LIN {X 0,Y 532.498,Z 413.718,A -85,B 0,C 180,E1 -4445.914,E2 -4445.914} C_VEL
LIN {X 0,Y 531.12,Z 406.108,A -85,B 0,C 180,E1 -4447.734,E2 -4447.734} C_VEL
LIN {X 0,Y 530.969,Z 405.349,A -85,B 0,C 180,E1 -4447.987,E2 -4447.987} C_VEL
LIN {X 0,Y 531.028,Z 405.342,A -85,B 0,C 180,E1 -4450.429,E2 -4450.429} C_VEL
LIN {X 0,Y 530.956,Z 405.351,A -85,B 0,C 180,E1 -4453.495,E2 -4453.495} C_VEL
LIN {X 0,Y 530.968,Z 405.348,A -85,B 0,C 180,E1 -4456.506,E2 -4456.506} C_VEL
LIN {X 0,Y 530.991,Z 405.345,A -85,B 0,C 180,E1 -4458.976,E2 -4458.976} C_VEL
LIN {X 0,Y 530.962,Z 405.348,A -85,B 0,C 180,E1 -4461.53,E2 -4461.53} C_VEL
LIN {X 0,Y 530.978,Z 405.348,A -85,B 0,C 180,E1 -4464.382,E2 -4464.382} C_VEL
LIN {X 0,Y 530.968,Z 405.345,A -85,B 0,C 180,E1 -4467.133,E2 -4467.133} C_VEL
LIN {X 0,Y 530.971,Z 405.348,A -85,B 0,C 180,E1 -4469.803,E2 -4469.803} C_VEL
LIN {X 0,Y 531.02,Z 405.341,A -85,B 0,C 180,E1 -4472.466,E2 -4472.466} C_VEL
LIN {X 0,Y 531.011,Z 405.342,A -85,B 0,C 180,E1 -4474.943,E2 -4474.943} C_VEL
LIN {X 0,Y 530.974,Z 405.347,A -85,B 0,C 180,E1 -4478.247,E2 -4478.247} C_VEL
LIN {X 0,Y 530.998,Z 405.345,A -85,B 0,C 180,E1 -4480.677,E2 -4480.677} C_VEL
LIN {X 0,Y 530.989,Z 405.344,A -85,B 0,C 180,E1 -4483.071,E2 -4483.071} C_VEL
LIN {X 0,Y 531.022,Z 405.34,A -85,B 0,C 180,E1 -4485.436,E2 -4485.436} C_VEL
LIN {X 0,Y 531.051,Z 405.337,A -85,B 0,C 180,E1 -4488.55,E2 -4488.55} C_VEL
LIN {X 0,Y 531.04,Z 405.34,A -85,B 0,C 180,E1 -4491.629,E2 -4491.629} C_VEL
LIN {X 0,Y 531.125,Z 405.329,A -85,B 0,C 180,E1 -4494.685,E2 -4494.685} C_VEL
LIN {X 0,Y 531.145,Z 405.325,A -85,B 0,C 180,E1 -4497.725,E2 -4497.725} C_VEL
LIN {X 0,Y 531.157,Z 405.323,A -85,B 0,C 180,E1 -4500.758,E2 -4500.758} C_VEL
LIN {X 0,Y 531.107,Z 405.328,A -85,B 0,C 180,E1 -4503.034,E2 -4503.034} C_VEL
LIN {X 0,Y 531.085,Z 405.333,A -85,B 0,C 180,E1 -4506.077,E2 -4506.077} C_VEL
LIN {X 0,Y 531.035,Z 405.339,A -85,B 0,C 180,E1 -4509.138,E2 -4509.138} C_VEL
LIN {X 0,Y 531.044,Z 405.339,A -85,B 0,C 180,E1 -4512.225,E2 -4512.225} C_VEL
LIN {X 0,Y 530.998,Z 405.344,A -85,B 0,C 180,E1 -4515.35,E2 -4515.35} C_VEL
LIN {X 0,Y 530.993,Z 405.345,A -85,B 0,C 180,E1 -4518.521,E2 -4518.521} C_VEL
LIN {X 0,Y 531.005,Z 405.343,A -85,B 0,C 180,E1 -4520.938,E2 -4520.938} C_VEL
LIN {X 0,Y 530.983,Z 405.346,A -85,B 0,C 180,E1 -4524.225,E2 -4524.225} C_VEL
LIN {X 0,Y 531.007,Z 405.341,A -85,B 0,C 180,E1 -4526.744,E2 -4526.744} C_VEL
LIN {X 0,Y 530.984,Z 405.345,A -85,B 0,C 180,E1 -4529.323,E2 -4529.323} C_VEL
LIN {X 0,Y 530.973,Z 405.347,A -85,B 0,C 180,E1 -4532.101,E2 -4532.101} C_VEL
LIN {X 0,Y 530.988,Z 405.345,A -85,B 0,C 180,E1 -4534.854,E2 -4534.854} C_VEL
LIN {X 0,Y 530.97,Z 405.347,A -85,B 0,C 180,E1 -4537.508,E2 -4537.508} C_VEL
LIN {X 0,Y 530.984,Z 405.345,A -85,B 0,C 180,E1 -4540.433,E2 -4540.433} C_VEL
LIN {X 0,Y 530.97,Z 405.348,A -85,B 0,C 180,E1 -4543.495,E2 -4543.495} C_VEL
LIN {X 0,Y 530.967,Z 405.348,A -85,B 0,C 180,E1 -4543.57,E2 -4543.57} C_VEL
LIN {X 0,Y 530.294,Z 405.432,A -85,B 0,C 180,E1 -4544.203,E2 -4544.203} C_VEL
LIN {X 0,Y 527.447,Z 405.786,A -85,B 0,C 180,E1 -4545.232,E2 -4545.232} C_VEL
LIN {X 0,Y 525.044,Z 406.087,A -85,B 0,C 180,E1 -4546.061,E2 -4546.061} C_VEL
LIN {X 0,Y 524.011,Z 406.214,A -85,B 0,C 180,E1 -4546.7,E2 -4546.7} C_VEL
LIN {X 0,Y 523.926,Z 406.224,A -85,B 0,C 180,E1 -4546.917,E2 -4546.917} C_VEL
LIN {X 0,Y 523.951,Z 406.223,A -85,B 0,C 180,E1 -4549.921,E2 -4549.921} C_VEL
LIN {X 0,Y 523.914,Z 406.224,A -85,B 0,C 180,E1 -4552.868,E2 -4552.868} C_VEL
LIN {X 0,Y 523.947,Z 406.223,A -85,B 0,C 180,E1 -4555.711,E2 -4555.711} C_VEL
LIN {X 0,Y 523.938,Z 406.224,A -85,B 0,C 180,E1 -4558.457,E2 -4558.457} C_VEL
LIN {X 0,Y 523.948,Z 406.222,A -85,B 0,C 180,E1 -4561.126,E2 -4561.126} C_VEL
LIN {X 0,Y 523.988,Z 406.218,A -85,B 0,C 180,E1 -4563.981,E2 -4563.981} C_VEL
LIN {X 0,Y 523.931,Z 406.224,A -85,B 0,C 180,E1 -4566.271,E2 -4566.271} C_VEL
LIN {X 0,Y 523.951,Z 406.221,A -85,B 0,C 180,E1 -4568.767,E2 -4568.767} C_VEL
LIN {X 0,Y 523.958,Z 406.22,A -85,B 0,C 180,E1 -4571.221,E2 -4571.221} C_VEL
LIN {X 0,Y 523.94,Z 406.223,A -85,B 0,C 180,E1 -4573.639,E2 -4573.639} C_VEL
LIN {X 0,Y 523.944,Z 406.224,A -85,B 0,C 180,E1 -4576.028,E2 -4576.028} C_VEL
LIN {X 0,Y 524.018,Z 406.214,A -85,B 0,C 180,E1 -4578.394,E2 -4578.394} C_VEL
LIN {X 0,Y 523.991,Z 406.288,A -85,B 0,C 180,E1 -4580.105,E2 -4580.105} C_VEL
LIN {X 0,Y 525.17,Z 411.277,A -85,B 0,C 180,E1 -4580.37,E2 -4580.37} C_VEL
LIN {X 0,Y 524.954,Z 423.401,A -85,B 0,C 180,E1 -4581.047,E2 -4581.047} C_VEL
LIN {X 0,Y 524.619,Z 435.388,A -85,B 0,C 180,E1 -4581.914,E2 -4581.914} C_VEL
LIN {X 0,Y 524.34,Z 445.661,A -85,B 0,C 180,E1 -4582.859,E2 -4582.859} C_VEL
LIN {X 0,Y 524.058,Z 454.306,A -85,B 0,C 180,E1 -4583.841,E2 -4583.841} C_VEL
LIN {X 0,Y 523.918,Z 461.363,A -85,B 0,C 180,E1 -4584.805,E2 -4584.805} C_VEL
LIN {X 0,Y 523.73,Z 468.234,A -85,B 0,C 180,E1 -4585.96,E2 -4585.96} C_VEL
LIN {X 0,Y 523.563,Z 474.542,A -85,B 0,C 180,E1 -4587.307,E2 -4587.307} C_VEL
LIN {X 0,Y 523.457,Z 479.837,A -85,B 0,C 180,E1 -4588.846,E2 -4588.846} C_VEL
LIN {X 0,Y 523.3,Z 482.596,A -85,B 0,C 180,E1 -4590,E2 -4590} C_VEL
LIN {X 0,Y 523.287,Z 483.993,A -85,B 0,C 180,E1 -4590.77,E2 -4590.77} C_VEL
LIN {X 0,Y 523.345,Z 485.482,A -85,B 0,C 180,E1 -4592.309,E2 -4592.309} C_VEL
LIN {X 0,Y 523.39,Z 485.664,A -85,B 0,C 180,E1 -4593.079,E2 -4593.079} C_VEL
LIN {X 0,Y 523.432,Z 485.43,A -85,B 0,C 180,E1 -4593.85,E2 -4593.85} C_VEL
LIN {X 0,Y 523.387,Z 483.874,A -85,B 0,C 180,E1 -4595.394,E2 -4595.394} C_VEL
LIN {X 0,Y 523.454,Z 480.665,A -85,B 0,C 180,E1 -4596.941,E2 -4596.941} C_VEL
LIN {X 0,Y 523.508,Z 477.124,A -85,B 0,C 180,E1 -4598.104,E2 -4598.104} C_VEL
LIN {X 0,Y 523.584,Z 472.411,A -85,B 0,C 180,E1 -4599.269,E2 -4599.269} C_VEL
LIN {X 0,Y 523.77,Z 466.518,A -85,B 0,C 180,E1 -4600.437,E2 -4600.437} C_VEL
LIN {X 0,Y 523.901,Z 459.174,A -85,B 0,C 180,E1 -4601.609,E2 -4601.609} C_VEL
LIN {X 0,Y 524.181,Z 449.879,A -85,B 0,C 180,E1 -4602.781,E2 -4602.781} C_VEL
LIN {X 0,Y 524.418,Z 440.224,A -85,B 0,C 180,E1 -4603.762,E2 -4603.762} C_VEL
LIN {X 0,Y 524.739,Z 430.634,A -85,B 0,C 180,E1 -4604.544,E2 -4604.544} C_VEL
LIN {X 0,Y 525.04,Z 420.234,A -85,B 0,C 180,E1 -4605.236,E2 -4605.236} C_VEL
LIN {X 0,Y 525.018,Z 410.197,A -85,B 0,C 180,E1 -4605.778,E2 -4605.778} C_VEL
LIN {X 0,Y 523.966,Z 406.223,A -85,B 0,C 180,E1 -4606.01,E2 -4606.01} C_VEL
LIN {X 0,Y 523.953,Z 406.22,A -85,B 0,C 180,E1 -4608.779,E2 -4608.779} C_VEL
LIN {X 0,Y 523.951,Z 406.215,A -85,B 0,C 180,E1 -4611.233,E2 -4611.233} C_VEL
LIN {X 0,Y 523.931,Z 406.222,A -85,B 0,C 180,E1 -4614.572,E2 -4614.572} C_VEL
LIN {X 0,Y 523.952,Z 406.214,A -85,B 0,C 180,E1 -4617.133,E2 -4617.133} C_VEL
LIN {X 0,Y 523.948,Z 406.217,A -85,B 0,C 180,E1 -4619.756,E2 -4619.756} C_VEL
LIN {X 0,Y 523.938,Z 406.221,A -85,B 0,C 180,E1 -4622.45,E2 -4622.45} C_VEL
LIN {X 0,Y 523.938,Z 406.216,A -85,B 0,C 180,E1 -4625.226,E2 -4625.226} C_VEL
LIN {X 0,Y 523.921,Z 406.226,A -85,B 0,C 180,E1 -4628.102,E2 -4628.102} C_VEL
LIN {X 0,Y 523.944,Z 406.215,A -85,B 0,C 180,E1 -4631.092,E2 -4631.092} C_VEL
LIN {X 0,Y 523.942,Z 406.222,A -85,B 0,C 180,E1 -4634.228,E2 -4634.228} C_VEL
LIN {X 0,Y 523.926,Z 406.217,A -85,B 0,C 180,E1 -4636.833,E2 -4636.833} C_VEL
LIN {X 0,Y 523.947,Z 406.215,A -85,B 0,C 180,E1 -4638.908,E2 -4638.908} C_VEL
LIN {X 0,Y 523.92,Z 406.226,A -85,B 0,C 180,E1 -4641.898,E2 -4641.898} C_VEL
LIN {X 0,Y 523.929,Z 406.217,A -85,B 0,C 180,E1 -4644.911,E2 -4644.911} C_VEL
LIN {X 0,Y 523.94,Z 406.221,A -85,B 0,C 180,E1 -4647.68,E2 -4647.68} C_VEL
LIN {X 0,Y 523.959,Z 406.213,A -85,B 0,C 180,E1 -4650.676,E2 -4650.676} C_VEL
LIN {X 0,Y 523.978,Z 406.218,A -85,B 0,C 180,E1 -4653.728,E2 -4653.728} C_VEL
LIN {X 0,Y 523.917,Z 406.221,A -85,B 0,C 180,E1 -4656.27,E2 -4656.27} C_VEL
LIN {X 0,Y 523.95,Z 406.214,A -85,B 0,C 180,E1 -4658.767,E2 -4658.767} C_VEL
LIN {X 0,Y 523.953,Z 406.216,A -85,B 0,C 180,E1 -4661.221,E2 -4661.221} C_VEL
LIN {X 0,Y 523.934,Z 406.224,A -85,B 0,C 180,E1 -4663.639,E2 -4663.639} C_VEL
LIN {X 0,Y 523.944,Z 406.221,A -85,B 0,C 180,E1 -4666.028,E2 -4666.028} C_VEL
LIN {X 0,Y 524.031,Z 406.283,A -85,B 0,C 180,E1 -4668.148,E2 -4668.148} C_VEL
LIN {X 0,Y 525.077,Z 411.361,A -85,B 0,C 180,E1 -4668.418,E2 -4668.418} C_VEL
LIN {X 0,Y 524.956,Z 421.94,A -85,B 0,C 180,E1 -4669.002,E2 -4669.002} C_VEL
LIN {X 0,Y 524.603,Z 433.114,A -85,B 0,C 180,E1 -4669.775,E2 -4669.775} C_VEL
LIN {X 0,Y 524.321,Z 444.072,A -85,B 0,C 180,E1 -4670.744,E2 -4670.744} C_VEL
LIN {X 0,Y 524.042,Z 452.907,A -85,B 0,C 180,E1 -4671.711,E2 -4671.711} C_VEL
LIN {X 0,Y 523.887,Z 460.199,A -85,B 0,C 180,E1 -4672.678,E2 -4672.678} C_VEL
LIN {X 0,Y 523.758,Z 467.369,A -85,B 0,C 180,E1 -4673.837,E2 -4673.837} C_VEL
LIN {X 0,Y 523.529,Z 473.11,A -85,B 0,C 180,E1 -4674.994,E2 -4674.994} C_VEL
LIN {X 0,Y 523.508,Z 477.591,A -85,B 0,C 180,E1 -4676.151,E2 -4676.151} C_VEL
LIN {X 0,Y 523.467,Z 479.958,A -85,B 0,C 180,E1 -4676.921,E2 -4676.921} C_VEL
LIN {X 0,Y 523.309,Z 483.443,A -85,B 0,C 180,E1 -4678.461,E2 -4678.461} C_VEL
LIN {X 0,Y 523.283,Z 484.58,A -85,B 0,C 180,E1 -4679.23,E2 -4679.23} C_VEL
LIN {X 0,Y 523.278,Z 485.616,A -85,B 0,C 180,E1 -4680.769,E2 -4680.769} C_VEL
LIN {X 0,Y 523.295,Z 485.594,A -85,B 0,C 180,E1 -4681.539,E2 -4681.539} C_VEL
LIN {X 0,Y 523.395,Z 484.295,A -85,B 0,C 180,E1 -4683.079,E2 -4683.079} C_VEL
LIN {X 0,Y 523.441,Z 483.112,A -85,B 0,C 180,E1 -4683.849,E2 -4683.849} C_VEL
LIN {X 0,Y 523.41,Z 480.522,A -85,B 0,C 180,E1 -4685.007,E2 -4685.007} C_VEL
LIN {X 0,Y 523.523,Z 476.921,A -85,B 0,C 180,E1 -4686.165,E2 -4686.165} C_VEL
LIN {X 0,Y 523.596,Z 472.211,A -85,B 0,C 180,E1 -4687.326,E2 -4687.326} C_VEL
LIN {X 0,Y 523.761,Z 466.229,A -85,B 0,C 180,E1 -4688.488,E2 -4688.488} C_VEL
LIN {X 0,Y 523.913,Z 460.139,A -85,B 0,C 180,E1 -4689.458,E2 -4689.458} C_VEL
LIN {X 0,Y 524.125,Z 452.795,A -85,B 0,C 180,E1 -4690.429,E2 -4690.429} C_VEL
LIN {X 0,Y 524.38,Z 443.885,A -85,B 0,C 180,E1 -4691.402,E2 -4691.402} C_VEL
LIN {X 0,Y 524.656,Z 432.719,A -85,B 0,C 180,E1 -4692.376,E2 -4692.376} C_VEL
LIN {X 0,Y 524.959,Z 421.283,A -85,B 0,C 180,E1 -4693.155,E2 -4693.155} C_VEL
LIN {X 0,Y 524.995,Z 410.363,A -85,B 0,C 180,E1 -4693.746,E2 -4693.746} C_VEL
LIN {X 0,Y 524.004,Z 406.214,A -85,B 0,C 180,E1 -4693.97,E2 -4693.97} C_VEL
LIN {X 0,Y 523.962,Z 406.221,A -85,B 0,C 180,E1 -4697.163,E2 -4697.163} C_VEL
LIN {X 0,Y 523.977,Z 406.221,A -85,B 0,C 180,E1 -4700.41,E2 -4700.41} C_VEL
LIN {X 0,Y 523.915,Z 406.228,A -85,B 0,C 180,E1 -4702.893,E2 -4702.893} C_VEL
LIN {X 0,Y 523.989,Z 406.217,A -85,B 0,C 180,E1 -4706.02,E2 -4706.02} C_VEL
LIN {X 0,Y 523.944,Z 406.222,A -85,B 0,C 180,E1 -4708.874,E2 -4708.874} C_VEL
LIN {X 0,Y 523.925,Z 406.225,A -85,B 0,C 180,E1 -4711.544,E2 -4711.544} C_VEL
LIN {X 0,Y 523.937,Z 406.224,A -85,B 0,C 180,E1 -4714.29,E2 -4714.29} C_VEL
LIN {X 0,Y 523.91,Z 406.226,A -85,B 0,C 180,E1 -4717.132,E2 -4717.132} C_VEL
LIN {X 0,Y 523.941,Z 406.222,A -85,B 0,C 180,E1 -4720.13,E2 -4720.13} C_VEL
LIN {X 0,Y 523.928,Z 406.223,A -85,B 0,C 180,E1 -4723.166,E2 -4723.166} C_VEL
LIN {X 0,Y 523.939,Z 406.22,A -85,B 0,C 180,E1 -4725.772,E2 -4725.772} C_VEL
LIN {X 0,Y 523.945,Z 406.222,A -85,B 0,C 180,E1 -4728.908,E2 -4728.908} C_VEL
LIN {X 0,Y 523.983,Z 406.405,A -85,B 0,C 180,E1 -4731.781,E2 -4731.781} C_VEL
LIN {X 0,Y 525.435,Z 413.966,A -85,B 0,C 180,E1 -4733.678,E2 -4733.678} C_VEL
LIN {X 0,Y 525.524,Z 419.21,A -85,B 0,C 180,E1 -4734.896,E2 -4734.896} C_VEL
LIN {X 0,Y 525.11,Z 433.663,A -85,B 0,C 180,E1 -4738.085,E2 -4738.085} C_VEL
LIN {X 0,Y 524.935,Z 446.556,A -85,B 0,C 180,E1 -4740.832,E2 -4740.832} C_VEL
LIN {X 0,Y 524.742,Z 461.045,A -85,B 0,C 180,E1 -4743.812,E2 -4743.812} C_VEL
LIN {X 0,Y 524.523,Z 476.503,A -85,B 0,C 180,E1 -4746.926,E2 -4746.926} C_VEL
LIN {X 0,Y 524.282,Z 490.939,A -85,B 0,C 180,E1 -4749.777,E2 -4749.777} C_VEL
LIN {X 0,Y 524.177,Z 504.983,A -85,B 0,C 180,E1 -4752.504,E2 -4752.504} C_VEL
LIN {X 0,Y 523.941,Z 522.326,A -85,B 0,C 180,E1 -4755.83,E2 -4755.83} C_VEL
LIN {X 0,Y 523.852,Z 524.508,A -85,B 0,C 180,E1 -4756.248,E2 -4756.248} C_VEL
LIN {X 0,Y 525.46,Z 535.938,A -85,B 0,C 180,E1 -4756.513,E2 -4756.513} C_VEL
LIN {X 0,Y 525.206,Z 548.7,A -85,B 0,C 180,E1 -4756.9,E2 -4756.9} C_VEL
LIN {X 0,Y 524.979,Z 561.165,A -85,B 0,C 180,E1 -4757.435,E2 -4757.435} C_VEL
LIN {X 0,Y 524.711,Z 573.14,A -85,B 0,C 180,E1 -4758.113,E2 -4758.113} C_VEL
LIN {X 0,Y 524.458,Z 583.898,A -85,B 0,C 180,E1 -4758.893,E2 -4758.893} C_VEL
LIN {X 0,Y 524.169,Z 593.595,A -85,B 0,C 180,E1 -4759.767,E2 -4759.767} C_VEL
LIN {X 0,Y 523.93,Z 602.411,A -85,B 0,C 180,E1 -4760.737,E2 -4760.737} C_VEL
LIN {X 0,Y 523.724,Z 611.003,A -85,B 0,C 180,E1 -4761.9,E2 -4761.9} C_VEL
LIN {X 0,Y 523.575,Z 617.867,A -85,B 0,C 180,E1 -4763.061,E2 -4763.061} C_VEL
LIN {X 0,Y 523.544,Z 623.365,A -85,B 0,C 180,E1 -4764.222,E2 -4764.222} C_VEL
LIN {X 0,Y 523.361,Z 627.676,A -85,B 0,C 180,E1 -4765.378,E2 -4765.378} C_VEL
LIN {X 0,Y 523.443,Z 629.957,A -85,B 0,C 180,E1 -4766.151,E2 -4766.151} C_VEL
LIN {X 0,Y 523.367,Z 631.806,A -85,B 0,C 180,E1 -4766.921,E2 -4766.921} C_VEL
LIN {X 0,Y 523.334,Z 633.193,A -85,B 0,C 180,E1 -4767.691,E2 -4767.691} C_VEL
LIN {X 0,Y 523.25,Z 634.785,A -85,B 0,C 180,E1 -4769.23,E2 -4769.23} C_VEL
LIN {X 0,Y 523.246,Z 635,A -85,B 0,C 180,E1 -4770,E2 -4770} C_VEL
LIN {X 0,Y 523.274,Z 634.184,A -85,B 0,C 180,E1 -4771.539,E2 -4771.539} C_VEL
LIN {X 0,Y 523.334,Z 633.196,A -85,B 0,C 180,E1 -4772.309,E2 -4772.309} C_VEL
LIN {X 0,Y 523.367,Z 631.81,A -85,B 0,C 180,E1 -4773.079,E2 -4773.079} C_VEL
LIN {X 0,Y 523.441,Z 628.896,A -85,B 0,C 180,E1 -4774.235,E2 -4774.235} C_VEL
LIN {X 0,Y 523.464,Z 624.948,A -85,B 0,C 180,E1 -4775.393,E2 -4775.393} C_VEL
LIN {X 0,Y 523.523,Z 619.727,A -85,B 0,C 180,E1 -4776.581,E2 -4776.581} C_VEL
LIN {X 0,Y 523.665,Z 613.467,A -85,B 0,C 180,E1 -4777.713,E2 -4777.713} C_VEL
LIN {X 0,Y 523.857,Z 605.478,A -85,B 0,C 180,E1 -4778.875,E2 -4778.875} C_VEL
LIN {X 0,Y 524.085,Z 597.334,A -85,B 0,C 180,E1 -4779.845,E2 -4779.845} C_VEL
LIN {X 0,Y 524.36,Z 587.395,A -85,B 0,C 180,E1 -4780.815,E2 -4780.815} C_VEL
LIN {X 0,Y 524.647,Z 577.521,A -85,B 0,C 180,E1 -4781.592,E2 -4781.592} C_VEL
LIN {X 0,Y 524.881,Z 566.042,A -85,B 0,C 180,E1 -4782.308,E2 -4782.308} C_VEL
LIN {X 0,Y 525.095,Z 553.693,A -85,B 0,C 180,E1 -4782.906,E2 -4782.906} C_VEL
LIN {X 0,Y 525.356,Z 540.547,A -85,B 0,C 180,E1 -4783.367,E2 -4783.367} C_VEL
LIN {X 0,Y 525.221,Z 533.738,A -85,B 0,C 180,E1 -4783.542,E2 -4783.542} C_VEL
LIN {X 0,Y 523.852,Z 524.533,A -85,B 0,C 180,E1 -4783.752,E2 -4783.752} C_VEL
LIN {X 0,Y 524.05,Z 509.933,A -85,B 0,C 180,E1 -4786.558,E2 -4786.558} C_VEL
LIN {X 0,Y 524.265,Z 495.307,A -85,B 0,C 180,E1 -4789.377,E2 -4789.377} C_VEL
LIN {X 0,Y 524.466,Z 481.727,A -85,B 0,C 180,E1 -4792.037,E2 -4792.037} C_VEL
LIN {X 0,Y 524.666,Z 466.125,A -85,B 0,C 180,E1 -4795.169,E2 -4795.169} C_VEL
LIN {X 0,Y 524.892,Z 451.487,A -85,B 0,C 180,E1 -4798.163,E2 -4798.163} C_VEL
LIN {X 0,Y 525.061,Z 437.633,A -85,B 0,C 180,E1 -4801.058,E2 -4801.058} C_VEL
LIN {X 0,Y 525.301,Z 424.197,A -85,B 0,C 180,E1 -4803.953,E2 -4803.953} C_VEL
LIN {X 0,Y 525.529,Z 414.817,A -85,B 0,C 180,E1 -4806.045,E2 -4806.045} C_VEL
LIN {X 0,Y 523.938,Z 406.224,A -85,B 0,C 180,E1 -4808.161,E2 -4808.161} C_VEL
LIN {X 0,Y 523.962,Z 406.221,A -85,B 0,C 180,E1 -4811.09,E2 -4811.09} C_VEL
LIN {X 0,Y 523.938,Z 406.224,A -85,B 0,C 180,E1 -4814.228,E2 -4814.228} C_VEL
LIN {X 0,Y 523.927,Z 406.228,A -85,B 0,C 180,E1 -4816.834,E2 -4816.834} C_VEL
LIN {X 0,Y 523.947,Z 406.223,A -85,B 0,C 180,E1 -4818.908,E2 -4818.908} C_VEL
LIN {X 0,Y 523.919,Z 406.225,A -85,B 0,C 180,E1 -4821.898,E2 -4821.898} C_VEL
LIN {X 0,Y 523.936,Z 406.222,A -85,B 0,C 180,E1 -4824.909,E2 -4824.909} C_VEL
LIN {X 0,Y 523.936,Z 406.223,A -85,B 0,C 180,E1 -4827.68,E2 -4827.68} C_VEL
LIN {X 0,Y 523.956,Z 406.221,A -85,B 0,C 180,E1 -4830.676,E2 -4830.676} C_VEL
LIN {X 0,Y 523.98,Z 406.217,A -85,B 0,C 180,E1 -4833.729,E2 -4833.729} C_VEL
LIN {X 0,Y 523.939,Z 406.225,A -85,B 0,C 180,E1 -4836.271,E2 -4836.271} C_VEL
LIN {X 0,Y 523.948,Z 406.221,A -85,B 0,C 180,E1 -4838.767,E2 -4838.767} C_VEL
LIN {X 0,Y 523.954,Z 406.219,A -85,B 0,C 180,E1 -4841.221,E2 -4841.221} C_VEL
LIN {X 0,Y 523.94,Z 406.222,A -85,B 0,C 180,E1 -4843.639,E2 -4843.639} C_VEL
LIN {X 0,Y 523.944,Z 406.224,A -85,B 0,C 180,E1 -4846.028,E2 -4846.028} C_VEL
LIN {X 0,Y 524.017,Z 406.214,A -85,B 0,C 180,E1 -4848.394,E2 -4848.394} C_VEL
LIN {X 0,Y 523.992,Z 406.217,A -85,B 0,C 180,E1 -4851.516,E2 -4851.516} C_VEL
LIN {X 0,Y 524.086,Z 406.206,A -85,B 0,C 180,E1 -4854.614,E2 -4854.614} C_VEL
LIN {X 0,Y 524.117,Z 406.201,A -85,B 0,C 180,E1 -4857.695,E2 -4857.695} C_VEL
LIN {X 0,Y 524.127,Z 406.198,A -85,B 0,C 180,E1 -4860.768,E2 -4860.768} C_VEL
LIN {X 0,Y 524.074,Z 406.205,A -85,B 0,C 180,E1 -4863.075,E2 -4863.075} C_VEL
LIN {X 0,Y 524.048,Z 406.209,A -85,B 0,C 180,E1 -4866.159,E2 -4866.159} C_VEL
LIN {X 0,Y 524.003,Z 406.214,A -85,B 0,C 180,E1 -4869.262,E2 -4869.262} C_VEL
LIN {X 0,Y 524.006,Z 406.214,A -85,B 0,C 180,E1 -4871.74,E2 -4871.74} C_VEL
LIN {X 0,Y 523.996,Z 406.215,A -85,B 0,C 180,E1 -4875.053,E2 -4875.053} C_VEL
LIN {X 0,Y 523.966,Z 406.22,A -85,B 0,C 180,E1 -4877.969,E2 -4877.969} C_VEL
LIN {X 0,Y 523.976,Z 406.218,A -85,B 0,C 180,E1 -4880.41,E2 -4880.41} C_VEL
LIN {X 0,Y 523.92,Z 406.225,A -85,B 0,C 180,E1 -4882.893,E2 -4882.893} C_VEL
LIN {X 0,Y 523.956,Z 406.221,A -85,B 0,C 180,E1 -4885.419,E2 -4885.419} C_VEL
LIN {X 0,Y 523.972,Z 406.219,A -85,B 0,C 180,E1 -4887.999,E2 -4887.999} C_VEL
LIN {X 0,Y 523.947,Z 406.221,A -85,B 0,C 180,E1 -4890.855,E2 -4890.855} C_VEL
LIN {X 0,Y 523.964,Z 406.221,A -85,B 0,C 180,E1 -4893.735,E2 -4893.735} C_VEL
LIN {X 0,Y 523.925,Z 406.224,A -85,B 0,C 180,E1 -4896.404,E2 -4896.404} C_VEL
LIN {X 0,Y 523.923,Z 406.224,A -85,B 0,C 180,E1 -4899.085,E2 -4899.085} C_VEL
LIN {X 0,Y 523.959,Z 406.221,A -85,B 0,C 180,E1 -4902.119,E2 -4902.119} C_VEL
LIN {X 0,Y 523.96,Z 406.22,A -85,B 0,C 180,E1 -4905.309,E2 -4905.309} C_VEL
LIN {X 0,Y 523.926,Z 406.224,A -85,B 0,C 180,E1 -4906.917,E2 -4906.917} C_VEL
LIN {X 0,Y 523.259,Z 406.308,A -85,B 0,C 180,E1 -4907.558,E2 -4907.558} C_VEL
LIN {X 0,Y 520.414,Z 406.662,A -85,B 0,C 180,E1 -4908.6,E2 -4908.6} C_VEL
LIN {X 0,Y 518.008,Z 406.963,A -85,B 0,C 180,E1 -4909.439,E2 -4909.439} C_VEL
LIN {X 0,Y 516.971,Z 407.092,A -85,B 0,C 180,E1 -4910.086,E2 -4910.086} C_VEL
LIN {X 0,Y 516.885,Z 407.101,A -85,B 0,C 180,E1 -4910.306,E2 -4910.306} C_VEL
LIN {X 0,Y 516.888,Z 407.102,A -85,B 0,C 180,E1 -4913.342,E2 -4913.342} C_VEL
LIN {X 0,Y 516.916,Z 407.098,A -85,B 0,C 180,E1 -4916.121,E2 -4916.121} C_VEL
LIN {X 0,Y 516.899,Z 407.1,A -85,B 0,C 180,E1 -4918.935,E2 -4918.935} C_VEL
LIN {X 0,Y 516.925,Z 407.097,A -85,B 0,C 180,E1 -4921.585,E2 -4921.585} C_VEL
LIN {X 0,Y 516.936,Z 407.095,A -85,B 0,C 180,E1 -4924.211,E2 -4924.211} C_VEL
LIN {X 0,Y 516.87,Z 407.102,A -85,B 0,C 180,E1 -4926.777,E2 -4926.777} C_VEL
LIN {X 0,Y 516.944,Z 407.095,A -85,B 0,C 180,E1 -4929.732,E2 -4929.732} C_VEL
LIN {X 0,Y 516.934,Z 407.095,A -85,B 0,C 180,E1 -4932.596,E2 -4932.596} C_VEL
LIN {X 0,Y 516.947,Z 407.095,A -85,B 0,C 180,E1 -4935.03,E2 -4935.03} C_VEL
LIN {X 0,Y 516.971,Z 407.091,A -85,B 0,C 180,E1 -4938.234,E2 -4938.234} C_VEL
LIN {X 0,Y 516.928,Z 407.168,A -85,B 0,C 180,E1 -4939.919,E2 -4939.919} C_VEL
LIN {X 0,Y 518.331,Z 413.084,A -85,B 0,C 180,E1 -4940.242,E2 -4940.242} C_VEL
LIN {X 0,Y 518.093,Z 425.044,A -85,B 0,C 180,E1 -4940.927,E2 -4940.927} C_VEL
LIN {X 0,Y 517.766,Z 435.721,A -85,B 0,C 180,E1 -4941.708,E2 -4941.708} C_VEL
LIN {X 0,Y 517.466,Z 444.979,A -85,B 0,C 180,E1 -4942.548,E2 -4942.548} C_VEL
LIN {X 0,Y 517.222,Z 454.167,A -85,B 0,C 180,E1 -4943.572,E2 -4943.572} C_VEL
LIN {X 0,Y 516.962,Z 462.643,A -85,B 0,C 180,E1 -4944.735,E2 -4944.735} C_VEL
LIN {X 0,Y 516.759,Z 469.461,A -85,B 0,C 180,E1 -4945.906,E2 -4945.906} C_VEL
LIN {X 0,Y 516.577,Z 475.707,A -85,B 0,C 180,E1 -4947.271,E2 -4947.271} C_VEL
LIN {X 0,Y 516.413,Z 479.828,A -85,B 0,C 180,E1 -4948.44,E2 -4948.44} C_VEL
LIN {X 0,Y 516.356,Z 481.999,A -85,B 0,C 180,E1 -4949.22,E2 -4949.22} C_VEL
LIN {X 0,Y 516.273,Z 485.054,A -85,B 0,C 180,E1 -4950.78,E2 -4950.78} C_VEL
LIN {X 0,Y 516.32,Z 486.518,A -85,B 0,C 180,E1 -4952.341,E2 -4952.341} C_VEL
LIN {X 0,Y 516.363,Z 486.668,A -85,B 0,C 180,E1 -4953.121,E2 -4953.121} C_VEL
LIN {X 0,Y 516.401,Z 486.421,A -85,B 0,C 180,E1 -4953.902,E2 -4953.902} C_VEL
LIN {X 0,Y 516.374,Z 484.823,A -85,B 0,C 180,E1 -4955.467,E2 -4955.467} C_VEL
LIN {X 0,Y 516.45,Z 481.566,A -85,B 0,C 180,E1 -4957.035,E2 -4957.035} C_VEL
LIN {X 0,Y 516.514,Z 477.984,A -85,B 0,C 180,E1 -4958.214,E2 -4958.214} C_VEL
LIN {X 0,Y 516.626,Z 473.262,A -85,B 0,C 180,E1 -4959.395,E2 -4959.395} C_VEL
LIN {X 0,Y 516.828,Z 467.318,A -85,B 0,C 180,E1 -4960.578,E2 -4960.578} C_VEL
LIN {X 0,Y 516.971,Z 459.906,A -85,B 0,C 180,E1 -4961.766,E2 -4961.766} C_VEL
LIN {X 0,Y 517.288,Z 450.519,A -85,B 0,C 180,E1 -4962.954,E2 -4962.954} C_VEL
LIN {X 0,Y 517.532,Z 440.784,A -85,B 0,C 180,E1 -4963.948,E2 -4963.948} C_VEL
LIN {X 0,Y 517.925,Z 429.786,A -85,B 0,C 180,E1 -4964.84,E2 -4964.84} C_VEL
LIN {X 0,Y 518.201,Z 419.429,A -85,B 0,C 180,E1 -4965.51,E2 -4965.51} C_VEL
LIN {X 0,Y 518.317,Z 413.367,A -85,B 0,C 180,E1 -4965.836,E2 -4965.836} C_VEL
LIN {X 0,Y 517.473,Z 409.196,A -85,B 0,C 180,E1 -4966.065,E2 -4966.065} C_VEL
LIN {X 0,Y 516.931,Z 407.1,A -85,B 0,C 180,E1 -4966.183,E2 -4966.183} C_VEL
LIN {X 0,Y 516.906,Z 407.095,A -85,B 0,C 180,E1 -4969.045,E2 -4969.045} C_VEL
LIN {X 0,Y 516.891,Z 407.095,A -85,B 0,C 180,E1 -4971.538,E2 -4971.538} C_VEL
LIN {X 0,Y 516.892,Z 407.102,A -85,B 0,C 180,E1 -4974.359,E2 -4974.359} C_VEL
LIN {X 0,Y 516.928,Z 407.093,A -85,B 0,C 180,E1 -4976.658,E2 -4976.658} C_VEL
LIN {X 0,Y 516.916,Z 407.091,A -85,B 0,C 180,E1 -4979.524,E2 -4979.524} C_VEL
LIN {X 0,Y 516.901,Z 407.097,A -85,B 0,C 180,E1 -4982.543,E2 -4982.543} C_VEL
LIN {X 0,Y 516.885,Z 407.094,A -85,B 0,C 180,E1 -4985.332,E2 -4985.332} C_VEL
LIN {X 0,Y 516.886,Z 407.1,A -85,B 0,C 180,E1 -4987.943,E2 -4987.943} C_VEL
LIN {X 0,Y 516.888,Z 407.095,A -85,B 0,C 180,E1 -4990.742,E2 -4990.742} C_VEL
LIN {X 0,Y 516.887,Z 407.095,A -85,B 0,C 180,E1 -4992.831,E2 -4992.831} C_VEL
LIN {X 0,Y 516.928,Z 407.089,A -85,B 0,C 180,E1 -4995.01,E2 -4995.01} C_VEL
LIN {X 0,Y 516.921,Z 407.094,A -85,B 0,C 180,E1 -4998.398,E2 -4998.398} C_VEL
LIN {X 0,Y 516.885,Z 407.095,A -85,B 0,C 180,E1 -5001.284,E2 -5001.284} C_VEL
LIN {X 0,Y 516.876,Z 407.101,A -85,B 0,C 180,E1 -5004.22,E2 -5004.22} C_VEL
LIN {X 0,Y 516.9,Z 407.093,A -85,B 0,C 180,E1 -5007.053,E2 -5007.053} C_VEL
LIN {X 0,Y 516.897,Z 407.101,A -85,B 0,C 180,E1 -5009.796,E2 -5009.796} C_VEL
LIN {X 0,Y 516.93,Z 407.09,A -85,B 0,C 180,E1 -5012.467,E2 -5012.467} C_VEL
LIN {X 0,Y 516.88,Z 407.095,A -85,B 0,C 180,E1 -5015.07,E2 -5015.07} C_VEL
LIN {X 0,Y 516.873,Z 407.102,A -85,B 0,C 180,E1 -5017.621,E2 -5017.621} C_VEL
LIN {X 0,Y 516.936,Z 407.092,A -85,B 0,C 180,E1 -5020.13,E2 -5020.13} C_VEL
LIN {X 0,Y 516.911,Z 407.091,A -85,B 0,C 180,E1 -5022.595,E2 -5022.595} C_VEL
LIN {X 0,Y 516.948,Z 407.088,A -85,B 0,C 180,E1 -5025.03,E2 -5025.03} C_VEL
LIN {X 0,Y 516.971,Z 407.142,A -85,B 0,C 180,E1 -5027.981,E2 -5027.981} C_VEL
LIN {X 0,Y 518.174,Z 412.313,A -85,B 0,C 180,E1 -5028.261,E2 -5028.261} C_VEL
LIN {X 0,Y 517.95,Z 424.416,A -85,B 0,C 180,E1 -5028.95,E2 -5028.95} C_VEL
LIN {X 0,Y 517.608,Z 436.424,A -85,B 0,C 180,E1 -5029.833,E2 -5029.833} C_VEL
LIN {X 0,Y 517.39,Z 444.997,A -85,B 0,C 180,E1 -5030.619,E2 -5030.619} C_VEL
LIN {X 0,Y 517.09,Z 453.845,A -85,B 0,C 180,E1 -5031.598,E2 -5031.598} C_VEL
LIN {X 0,Y 516.921,Z 461.153,A -85,B 0,C 180,E1 -5032.579,E2 -5032.579} C_VEL
LIN {X 0,Y 516.762,Z 468.314,A -85,B 0,C 180,E1 -5033.754,E2 -5033.754} C_VEL
LIN {X 0,Y 516.528,Z 474.065,A -85,B 0,C 180,E1 -5034.926,E2 -5034.926} C_VEL
LIN {X 0,Y 516.493,Z 478.569,A -85,B 0,C 180,E1 -5036.099,E2 -5036.099} C_VEL
LIN {X 0,Y 516.449,Z 480.958,A -85,B 0,C 180,E1 -5036.88,E2 -5036.88} C_VEL
LIN {X 0,Y 516.305,Z 484.455,A -85,B 0,C 180,E1 -5038.44,E2 -5038.44} C_VEL
LIN {X 0,Y 516.269,Z 485.586,A -85,B 0,C 180,E1 -5039.22,E2 -5039.22} C_VEL
LIN {X 0,Y 516.265,Z 486.643,A -85,B 0,C 180,E1 -5040.78,E2 -5040.78} C_VEL
LIN {X 0,Y 516.292,Z 486.602,A -85,B 0,C 180,E1 -5041.56,E2 -5041.56} C_VEL
LIN {X 0,Y 516.376,Z 485.315,A -85,B 0,C 180,E1 -5043.121,E2 -5043.121} C_VEL
LIN {X 0,Y 516.421,Z 484.109,A -85,B 0,C 180,E1 -5043.902,E2 -5043.902} C_VEL
LIN {X 0,Y 516.424,Z 481.506,A -85,B 0,C 180,E1 -5045.075,E2 -5045.075} C_VEL
LIN {X 0,Y 516.541,Z 477.892,A -85,B 0,C 180,E1 -5046.249,E2 -5046.249} C_VEL
LIN {X 0,Y 516.622,Z 473.182,A -85,B 0,C 180,E1 -5047.425,E2 -5047.425} C_VEL
LIN {X 0,Y 516.809,Z 467.185,A -85,B 0,C 180,E1 -5048.603,E2 -5048.603} C_VEL
LIN {X 0,Y 516.979,Z 459.707,A -85,B 0,C 180,E1 -5049.784,E2 -5049.784} C_VEL
LIN {X 0,Y 517.287,Z 450.324,A -85,B 0,C 180,E1 -5050.965,E2 -5050.965} C_VEL
LIN {X 0,Y 517.514,Z 441.149,A -85,B 0,C 180,E1 -5051.894,E2 -5051.894} C_VEL
LIN {X 0,Y 517.862,Z 430.79,A -85,B 0,C 180,E1 -5052.74,E2 -5052.74} C_VEL
LIN {X 0,Y 518.099,Z 420.271,A -85,B 0,C 180,E1 -5053.432,E2 -5053.432} C_VEL
LIN {X 0,Y 518.18,Z 411.907,A -85,B 0,C 180,E1 -5053.88,E2 -5053.88} C_VEL
LIN {X 0,Y 516.959,Z 407.092,A -85,B 0,C 180,E1 -5054.139,E2 -5054.139} C_VEL
LIN {X 0,Y 516.912,Z 407.102,A -85,B 0,C 180,E1 -5057.404,E2 -5057.404} C_VEL
LIN {X 0,Y 516.944,Z 407.099,A -85,B 0,C 180,E1 -5060.268,E2 -5060.268} C_VEL
LIN {X 0,Y 516.864,Z 407.105,A -85,B 0,C 180,E1 -5063.224,E2 -5063.224} C_VEL
LIN {X 0,Y 516.947,Z 407.093,A -85,B 0,C 180,E1 -5066.196,E2 -5066.196} C_VEL
LIN {X 0,Y 516.926,Z 407.094,A -85,B 0,C 180,E1 -5069.304,E2 -5069.304} C_VEL
LIN {X 0,Y 516.899,Z 407.1,A -85,B 0,C 180,E1 -5072.543,E2 -5072.543} C_VEL
LIN {X 0,Y 516.87,Z 407.104,A -85,B 0,C 180,E1 -5075.33,E2 -5075.33} C_VEL
LIN {X 0,Y 516.883,Z 407.1,A -85,B 0,C 180,E1 -5077.943,E2 -5077.943} C_VEL
LIN {X 0,Y 516.887,Z 407.101,A -85,B 0,C 180,E1 -5080.741,E2 -5080.741} C_VEL
LIN {X 0,Y 516.908,Z 407.099,A -85,B 0,C 180,E1 -5082.829,E2 -5082.829} C_VEL
LIN {X 0,Y 516.926,Z 407.097,A -85,B 0,C 180,E1 -5085.01,E2 -5085.01} C_VEL
LIN {X 0,Y 516.918,Z 407.098,A -85,B 0,C 180,E1 -5088.398,E2 -5088.398} C_VEL
LIN {X 0,Y 516.921,Z 407.129,A -85,B 0,C 180,E1 -5091.485,E2 -5091.485} C_VEL
LIN {X 0,Y 518.527,Z 415.517,A -85,B 0,C 180,E1 -5093.631,E2 -5093.631} C_VEL
LIN {X 0,Y 518.593,Z 420.692,A -85,B 0,C 180,E1 -5094.844,E2 -5094.844} C_VEL
LIN {X 0,Y 518.182,Z 433.144,A -85,B 0,C 180,E1 -5097.642,E2 -5097.642} C_VEL
LIN {X 0,Y 517.97,Z 446.325,A -85,B 0,C 180,E1 -5100.512,E2 -5100.512} C_VEL
LIN {X 0,Y 517.708,Z 461.202,A -85,B 0,C 180,E1 -5103.633,E2 -5103.633} C_VEL
LIN {X 0,Y 517.488,Z 475.658,A -85,B 0,C 180,E1 -5106.594,E2 -5106.594} C_VEL
LIN {X 0,Y 517.286,Z 489.175,A -85,B 0,C 180,E1 -5109.314,E2 -5109.314} C_VEL
LIN {X 0,Y 517.107,Z 504.397,A -85,B 0,C 180,E1 -5112.332,E2 -5112.332} C_VEL
LIN {X 0,Y 516.863,Z 520.243,A -85,B 0,C 180,E1 -5115.43,E2 -5115.43} C_VEL
LIN {X 0,Y 516.798,Z 523.459,A -85,B 0,C 180,E1 -5116.057,E2 -5116.057} C_VEL
LIN {X 0,Y 518.494,Z 536.746,A -85,B 0,C 180,E1 -5116.378,E2 -5116.378} C_VEL
LIN {X 0,Y 518.187,Z 550.286,A -85,B 0,C 180,E1 -5116.819,E2 -5116.819} C_VEL
LIN {X 0,Y 517.943,Z 562.076,A -85,B 0,C 180,E1 -5117.361,E2 -5117.361} C_VEL
LIN {X 0,Y 517.657,Z 573.708,A -85,B 0,C 180,E1 -5118.059,E2 -5118.059} C_VEL
LIN {X 0,Y 517.36,Z 585.318,A -85,B 0,C 180,E1 -5118.937,E2 -5118.937} C_VEL
LIN {X 0,Y 517.058,Z 594.786,A -85,B 0,C 180,E1 -5119.822,E2 -5119.822} C_VEL
LIN {X 0,Y 516.825,Z 603.443,A -85,B 0,C 180,E1 -5120.806,E2 -5120.806} C_VEL
LIN {X 0,Y 516.617,Z 611.901,A -85,B 0,C 180,E1 -5121.984,E2 -5121.984} C_VEL
LIN {X 0,Y 516.507,Z 617.696,A -85,B 0,C 180,E1 -5122.966,E2 -5122.966} C_VEL
LIN {X 0,Y 516.454,Z 623.31,A -85,B 0,C 180,E1 -5124.142,E2 -5124.142} C_VEL
LIN {X 0,Y 516.271,Z 627.662,A -85,B 0,C 180,E1 -5125.315,E2 -5125.315} C_VEL
LIN {X 0,Y 516.354,Z 629.956,A -85,B 0,C 180,E1 -5126.098,E2 -5126.098} C_VEL
LIN {X 0,Y 516.282,Z 631.806,A -85,B 0,C 180,E1 -5126.878,E2 -5126.878} C_VEL
LIN {X 0,Y 516.261,Z 633.192,A -85,B 0,C 180,E1 -5127.659,E2 -5127.659} C_VEL
LIN {X 0,Y 516.16,Z 634.785,A -85,B 0,C 180,E1 -5129.22,E2 -5129.22} C_VEL
LIN {X 0,Y 516.154,Z 635,A -85,B 0,C 180,E1 -5130,E2 -5130} C_VEL
LIN {X 0,Y 516.192,Z 634.183,A -85,B 0,C 180,E1 -5131.56,E2 -5131.56} C_VEL
LIN {X 0,Y 516.26,Z 633.195,A -85,B 0,C 180,E1 -5132.34,E2 -5132.34} C_VEL
LIN {X 0,Y 516.282,Z 631.81,A -85,B 0,C 180,E1 -5133.121,E2 -5133.121} C_VEL
LIN {X 0,Y 516.343,Z 628.891,A -85,B 0,C 180,E1 -5134.293,E2 -5134.293} C_VEL
LIN {X 0,Y 516.405,Z 624.913,A -85,B 0,C 180,E1 -5135.466,E2 -5135.466} C_VEL
LIN {X 0,Y 516.479,Z 618.943,A -85,B 0,C 180,E1 -5136.797,E2 -5136.797} C_VEL
LIN {X 0,Y 516.617,Z 611.905,A -85,B 0,C 180,E1 -5138.015,E2 -5138.015} C_VEL
LIN {X 0,Y 516.825,Z 603.449,A -85,B 0,C 180,E1 -5139.194,E2 -5139.194} C_VEL
LIN {X 0,Y 517.058,Z 594.796,A -85,B 0,C 180,E1 -5140.177,E2 -5140.177} C_VEL
LIN {X 0,Y 517.402,Z 584.138,A -85,B 0,C 180,E1 -5141.161,E2 -5141.161} C_VEL
LIN {X 0,Y 517.65,Z 572.583,A -85,B 0,C 180,E1 -5142.019,E2 -5142.019} C_VEL
LIN {X 0,Y 517.968,Z 562.098,A -85,B 0,C 180,E1 -5142.638,E2 -5142.638} C_VEL
LIN {X 0,Y 518.197,Z 550.302,A -85,B 0,C 180,E1 -5143.18,E2 -5143.18} C_VEL
LIN {X 0,Y 518.463,Z 536.765,A -85,B 0,C 180,E1 -5143.622,E2 -5143.622} C_VEL
LIN {X 0,Y 516.797,Z 523.565,A -85,B 0,C 180,E1 -5143.943,E2 -5143.943} C_VEL
LIN {X 0,Y 517.078,Z 506.973,A -85,B 0,C 180,E1 -5147.195,E2 -5147.195} C_VEL
LIN {X 0,Y 517.285,Z 490.741,A -85,B 0,C 180,E1 -5150.371,E2 -5150.371} C_VEL
LIN {X 0,Y 517.481,Z 475.734,A -85,B 0,C 180,E1 -5153.406,E2 -5153.406} C_VEL
LIN {X 0,Y 517.724,Z 461.28,A -85,B 0,C 180,E1 -5156.371,E2 -5156.371} C_VEL
LIN {X 0,Y 517.926,Z 447.531,A -85,B 0,C 180,E1 -5159.242,E2 -5159.242} C_VEL
LIN {X 0,Y 518.16,Z 434.92,A -85,B 0,C 180,E1 -5161.936,E2 -5161.936} C_VEL
LIN {X 0,Y 518.508,Z 420.389,A -85,B 0,C 180,E1 -5165.153,E2 -5165.153} C_VEL
LIN {X 0,Y 518.454,Z 415.098,A -85,B 0,C 180,E1 -5166.374,E2 -5166.374} C_VEL
LIN {X 0,Y 516.896,Z 407.101,A -85,B 0,C 180,E1 -5168.412,E2 -5168.412} C_VEL
LIN {X 0,Y 516.905,Z 407.1,A -85,B 0,C 180,E1 -5170.74,E2 -5170.74} C_VEL
LIN {X 0,Y 516.883,Z 407.104,A -85,B 0,C 180,E1 -5173.903,E2 -5173.903} C_VEL
LIN {X 0,Y 516.884,Z 407.102,A -85,B 0,C 180,E1 -5176.107,E2 -5176.107} C_VEL
LIN {X 0,Y 516.919,Z 407.097,A -85,B 0,C 180,E1 -5178.398,E2 -5178.398} C_VEL
LIN {X 0,Y 516.885,Z 407.101,A -85,B 0,C 180,E1 -5181.284,E2 -5181.284} C_VEL
LIN {X 0,Y 516.889,Z 407.102,A -85,B 0,C 180,E1 -5184.221,E2 -5184.221} C_VEL
LIN {X 0,Y 516.896,Z 407.098,A -85,B 0,C 180,E1 -5187.053,E2 -5187.053} C_VEL
LIN {X 0,Y 516.894,Z 407.101,A -85,B 0,C 180,E1 -5189.796,E2 -5189.796} C_VEL
LIN {X 0,Y 516.933,Z 407.095,A -85,B 0,C 180,E1 -5192.468,E2 -5192.468} C_VEL
LIN {X 0,Y 516.914,Z 407.098,A -85,B 0,C 180,E1 -5195.072,E2 -5195.072} C_VEL
LIN {X 0,Y 516.888,Z 407.103,A -85,B 0,C 180,E1 -5198.462,E2 -5198.462} C_VEL
LIN {X 0,Y 516.905,Z 407.098,A -85,B 0,C 180,E1 -5200.955,E2 -5200.955} C_VEL
LIN {X 0,Y 516.917,Z 407.096,A -85,B 0,C 180,E1 -5203.41,E2 -5203.41} C_VEL
LIN {X 0,Y 516.898,Z 407.1,A -85,B 0,C 180,E1 -5205.834,E2 -5205.834} C_VEL
LIN {X 0,Y 517.007,Z 407.088,A -85,B 0,C 180,E1 -5208.235,E2 -5208.235} C_VEL
LIN {X 0,Y 516.96,Z 407.091,A -85,B 0,C 180,E1 -5211.4,E2 -5211.4} C_VEL
LIN {X 0,Y 517.013,Z 407.087,A -85,B 0,C 180,E1 -5213.757,E2 -5213.757} C_VEL
LIN {X 0,Y 517.089,Z 407.076,A -85,B 0,C 180,E1 -5217.663,E2 -5217.663} C_VEL
LIN {X 0,Y 517.098,Z 407.074,A -85,B 0,C 180,E1 -5220.779,E2 -5220.779} C_VEL
LIN {X 0,Y 517.015,Z 407.084,A -85,B 0,C 180,E1 -5223.117,E2 -5223.117} C_VEL
LIN {X 0,Y 517.012,Z 407.086,A -85,B 0,C 180,E1 -5226.243,E2 -5226.243} C_VEL
LIN {X 0,Y 516.958,Z 407.092,A -85,B 0,C 180,E1 -5229.389,E2 -5229.389} C_VEL
LIN {X 0,Y 516.955,Z 407.093,A -85,B 0,C 180,E1 -5231.808,E2 -5231.808} C_VEL
LIN {X 0,Y 516.947,Z 407.093,A -85,B 0,C 180,E1 -5235.147,E2 -5235.147} C_VEL
LIN {X 0,Y 516.928,Z 407.096,A -85,B 0,C 180,E1 -5238.222,E2 -5238.222} C_VEL
LIN {X 0,Y 516.916,Z 407.098,A -85,B 0,C 180,E1 -5240.702,E2 -5240.702} C_VEL
LIN {X 0,Y 516.914,Z 407.099,A -85,B 0,C 180,E1 -5244.072,E2 -5244.072} C_VEL
LIN {X 0,Y 516.928,Z 407.095,A -85,B 0,C 180,E1 -5246.658,E2 -5246.658} C_VEL
LIN {X 0,Y 516.913,Z 407.099,A -85,B 0,C 180,E1 -5249.524,E2 -5249.524} C_VEL
LIN {X 0,Y 516.9,Z 407.1,A -85,B 0,C 180,E1 -5252.544,E2 -5252.544} C_VEL
LIN {X 0,Y 516.884,Z 407.101,A -85,B 0,C 180,E1 -5255.332,E2 -5255.332} C_VEL
LIN {X 0,Y 516.884,Z 407.103,A -85,B 0,C 180,E1 -5257.943,E2 -5257.943} C_VEL
LIN {X 0,Y 516.887,Z 407.099,A -85,B 0,C 180,E1 -5260.742,E2 -5260.742} C_VEL
LIN {X 0,Y 516.908,Z 407.097,A -85,B 0,C 180,E1 -5262.829,E2 -5262.829} C_VEL
LIN {X 0,Y 516.926,Z 407.096,A -85,B 0,C 180,E1 -5265.01,E2 -5265.01} C_VEL
LIN {X 0,Y 516.921,Z 407.096,A -85,B 0,C 180,E1 -5268.398,E2 -5268.398} C_VEL
LIN {X 0,Y 516.885,Z 407.101,A -85,B 0,C 180,E1 -5270.306,E2 -5270.306} C_VEL
LIN {X 0,Y 516.215,Z 407.185,A -85,B 0,C 180,E1 -5270.956,E2 -5270.956} C_VEL
LIN {X 0,Y 513.37,Z 407.541,A -85,B 0,C 180,E1 -5272.012,E2 -5272.012} C_VEL
LIN {X 0,Y 510.962,Z 407.842,A -85,B 0,C 180,E1 -5272.862,E2 -5272.862} C_VEL
LIN {X 0,Y 509.922,Z 407.97,A -85,B 0,C 180,E1 -5273.518,E2 -5273.518} C_VEL
LIN {X 0,Y 509.834,Z 407.98,A -85,B 0,C 180,E1 -5273.741,E2 -5273.741} C_VEL
LIN {X 0,Y 509.867,Z 407.975,A -85,B 0,C 180,E1 -5276.54,E2 -5276.54} C_VEL
LIN {X 0,Y 509.855,Z 407.977,A -85,B 0,C 180,E1 -5279.335,E2 -5279.335} C_VEL
LIN {X 0,Y 509.898,Z 407.972,A -85,B 0,C 180,E1 -5282.055,E2 -5282.055} C_VEL
LIN {X 0,Y 509.88,Z 407.972,A -85,B 0,C 180,E1 -5284.704,E2 -5284.704} C_VEL
LIN {X 0,Y 509.831,Z 407.982,A -85,B 0,C 180,E1 -5287.458,E2 -5287.458} C_VEL
LIN {X 0,Y 509.922,Z 407.969,A -85,B 0,C 180,E1 -5289.845,E2 -5289.845} C_VEL
LIN {X 0,Y 509.888,Z 407.973,A -85,B 0,C 180,E1 -5293.175,E2 -5293.175} C_VEL
LIN {X 0,Y 509.868,Z 407.976,A -85,B 0,C 180,E1 -5295.634,E2 -5295.634} C_VEL
LIN {X 0,Y 509.919,Z 407.969,A -85,B 0,C 180,E1 -5298.875,E2 -5298.875} C_VEL
LIN {X 0,Y 509.879,Z 408.065,A -85,B 0,C 180,E1 -5299.728,E2 -5299.728} C_VEL
LIN {X 0,Y 511.248,Z 413.031,A -85,B 0,C 180,E1 -5300.006,E2 -5300.006} C_VEL
LIN {X 0,Y 511.387,Z 418.604,A -85,B 0,C 180,E1 -5300.308,E2 -5300.308} C_VEL
LIN {X 0,Y 511.134,Z 429.511,A -85,B 0,C 180,E1 -5301.002,E2 -5301.002} C_VEL
LIN {X 0,Y 510.699,Z 440.656,A -85,B 0,C 180,E1 -5301.891,E2 -5301.891} C_VEL
LIN {X 0,Y 510.41,Z 450.459,A -85,B 0,C 180,E1 -5302.882,E2 -5302.882} C_VEL
LIN {X 0,Y 510.176,Z 458.473,A -85,B 0,C 180,E1 -5303.872,E2 -5303.872} C_VEL
LIN {X 0,Y 509.926,Z 466.323,A -85,B 0,C 180,E1 -5305.059,E2 -5305.059} C_VEL
LIN {X 0,Y 509.706,Z 471.665,A -85,B 0,C 180,E1 -5306.047,E2 -5306.047} C_VEL
LIN {X 0,Y 509.59,Z 476.872,A -85,B 0,C 180,E1 -5307.233,E2 -5307.233} C_VEL
LIN {X 0,Y 509.427,Z 480.954,A -85,B 0,C 180,E1 -5308.419,E2 -5308.419} C_VEL
LIN {X 0,Y 509.361,Z 483.115,A -85,B 0,C 180,E1 -5309.21,E2 -5309.21} C_VEL
LIN {X 0,Y 509.258,Z 486.116,A -85,B 0,C 180,E1 -5310.791,E2 -5310.791} C_VEL
LIN {X 0,Y 509.296,Z 487.554,A -85,B 0,C 180,E1 -5312.373,E2 -5312.373} C_VEL
LIN {X 0,Y 509.37,Z 487.408,A -85,B 0,C 180,E1 -5313.956,E2 -5313.956} C_VEL
LIN {X 0,Y 509.364,Z 485.771,A -85,B 0,C 180,E1 -5315.543,E2 -5315.543} C_VEL
LIN {X 0,Y 509.408,Z 483.727,A -85,B 0,C 180,E1 -5316.612,E2 -5316.612} C_VEL
LIN {X 0,Y 509.468,Z 480.183,A -85,B 0,C 180,E1 -5317.929,E2 -5317.929} C_VEL
LIN {X 0,Y 509.623,Z 475.833,A -85,B 0,C 180,E1 -5319.125,E2 -5319.125} C_VEL
LIN {X 0,Y 509.832,Z 469.206,A -85,B 0,C 180,E1 -5320.524,E2 -5320.524} C_VEL
LIN {X 0,Y 510.017,Z 461.99,A -85,B 0,C 180,E1 -5321.725,E2 -5321.725} C_VEL
LIN {X 0,Y 510.276,Z 454.559,A -85,B 0,C 180,E1 -5322.731,E2 -5322.731} C_VEL
LIN {X 0,Y 510.554,Z 445.547,A -85,B 0,C 180,E1 -5323.737,E2 -5323.737} C_VEL
LIN {X 0,Y 510.924,Z 435.477,A -85,B 0,C 180,E1 -5324.641,E2 -5324.641} C_VEL
LIN {X 0,Y 511.239,Z 424.775,A -85,B 0,C 180,E1 -5325.413,E2 -5325.413} C_VEL
LIN {X 0,Y 511.36,Z 413.538,A -85,B 0,C 180,E1 -5326.057,E2 -5326.057} C_VEL
LIN {X 0,Y 509.876,Z 407.978,A -85,B 0,C 180,E1 -5326.388,E2 -5326.388} C_VEL
LIN {X 0,Y 509.867,Z 407.971,A -85,B 0,C 180,E1 -5329.319,E2 -5329.319} C_VEL
LIN {X 0,Y 509.827,Z 407.977,A -85,B 0,C 180,E1 -5331.851,E2 -5331.851} C_VEL
LIN {X 0,Y 509.848,Z 407.977,A -85,B 0,C 180,E1 -5334.524,E2 -5334.524} C_VEL
LIN {X 0,Y 509.887,Z 407.967,A -85,B 0,C 180,E1 -5337.056,E2 -5337.056} C_VEL
LIN {X 0,Y 509.863,Z 407.971,A -85,B 0,C 180,E1 -5339.751,E2 -5339.751} C_VEL
LIN {X 0,Y 509.878,Z 407.969,A -85,B 0,C 180,E1 -5342.774,E2 -5342.774} C_VEL
LIN {X 0,Y 509.845,Z 407.973,A -85,B 0,C 180,E1 -5345.581,E2 -5345.581} C_VEL
LIN {X 0,Y 509.855,Z 407.976,A -85,B 0,C 180,E1 -5348.338,E2 -5348.338} C_VEL
LIN {X 0,Y 509.86,Z 407.97,A -85,B 0,C 180,E1 -5351.426,E2 -5351.426} C_VEL
LIN {X 0,Y 509.862,Z 407.971,A -85,B 0,C 180,E1 -5354.668,E2 -5354.668} C_VEL
LIN {X 0,Y 509.863,Z 407.977,A -85,B 0,C 180,E1 -5358.103,E2 -5358.103} C_VEL
LIN {X 0,Y 509.851,Z 407.972,A -85,B 0,C 180,E1 -5360.648,E2 -5360.648} C_VEL
LIN {X 0,Y 509.829,Z 407.978,A -85,B 0,C 180,E1 -5363.647,E2 -5363.647} C_VEL
LIN {X 0,Y 509.864,Z 407.97,A -85,B 0,C 180,E1 -5366.539,E2 -5366.539} C_VEL
LIN {X 0,Y 509.85,Z 407.972,A -85,B 0,C 180,E1 -5369.334,E2 -5369.334} C_VEL
LIN {X 0,Y 509.896,Z 407.971,A -85,B 0,C 180,E1 -5372.054,E2 -5372.054} C_VEL
LIN {X 0,Y 509.845,Z 407.971,A -85,B 0,C 180,E1 -5374.702,E2 -5374.702} C_VEL
LIN {X 0,Y 509.831,Z 407.977,A -85,B 0,C 180,E1 -5377.458,E2 -5377.458} C_VEL
LIN {X 0,Y 509.922,Z 407.97,A -85,B 0,C 180,E1 -5379.845,E2 -5379.845} C_VEL
LIN {X 0,Y 509.877,Z 407.969,A -85,B 0,C 180,E1 -5383.174,E2 -5383.174} C_VEL
LIN {X 0,Y 509.869,Z 407.977,A -85,B 0,C 180,E1 -5385.634,E2 -5385.634} C_VEL
LIN {X 0,Y 509.926,Z 407.97,A -85,B 0,C 180,E1 -5387.801,E2 -5387.801} C_VEL
LIN {X 0,Y 511.268,Z 413.264,A -85,B 0,C 180,E1 -5388.1,E2 -5388.1} C_VEL
LIN {X 0,Y 511.042,Z 425.383,A -85,B 0,C 180,E1 -5388.805,E2 -5388.805} C_VEL
LIN {X 0,Y 510.703,Z 436.109,A -85,B 0,C 180,E1 -5389.594,E2 -5389.594} C_VEL
LIN {X 0,Y 510.469,Z 445.916,A -85,B 0,C 180,E1 -5390.49,E2 -5390.49} C_VEL
LIN {X 0,Y 510.139,Z 454.779,A -85,B 0,C 180,E1 -5391.483,E2 -5391.483} C_VEL
LIN {X 0,Y 509.915,Z 463.403,A -85,B 0,C 180,E1 -5392.675,E2 -5392.675} C_VEL
LIN {X 0,Y 509.767,Z 470.331,A -85,B 0,C 180,E1 -5393.866,E2 -5393.866} C_VEL
LIN {X 0,Y 509.499,Z 476.637,A -85,B 0,C 180,E1 -5395.252,E2 -5395.252} C_VEL
LIN {X 0,Y 509.52,Z 480.766,A -85,B 0,C 180,E1 -5396.441,E2 -5396.441} C_VEL
LIN {X 0,Y 509.333,Z 483.881,A -85,B 0,C 180,E1 -5397.627,E2 -5397.627} C_VEL
LIN {X 0,Y 509.299,Z 485.449,A -85,B 0,C 180,E1 -5398.418,E2 -5398.418} C_VEL
LIN {X 0,Y 509.254,Z 486.587,A -85,B 0,C 180,E1 -5399.209,E2 -5399.209} C_VEL
LIN {X 0,Y 509.25,Z 487.646,A -85,B 0,C 180,E1 -5400.791,E2 -5400.791} C_VEL
LIN {X 0,Y 509.286,Z 487.61,A -85,B 0,C 180,E1 -5401.581,E2 -5401.581} C_VEL
LIN {X 0,Y 509.308,Z 487.17,A -85,B 0,C 180,E1 -5402.372,E2 -5402.372} C_VEL
LIN {X 0,Y 509.402,Z 485.106,A -85,B 0,C 180,E1 -5403.955,E2 -5403.955} C_VEL
LIN {X 0,Y 509.436,Z 482.489,A -85,B 0,C 180,E1 -5405.145,E2 -5405.145} C_VEL
LIN {X 0,Y 509.56,Z 478.863,A -85,B 0,C 180,E1 -5406.335,E2 -5406.335} C_VEL
LIN {X 0,Y 509.653,Z 474.134,A -85,B 0,C 180,E1 -5407.527,E2 -5407.527} C_VEL
LIN {X 0,Y 509.86,Z 468.136,A -85,B 0,C 180,E1 -5408.721,E2 -5408.721} C_VEL
LIN {X 0,Y 510.041,Z 460.59,A -85,B 0,C 180,E1 -5409.918,E2 -5409.918} C_VEL
LIN {X 0,Y 510.357,Z 452.861,A -85,B 0,C 180,E1 -5410.915,E2 -5410.915} C_VEL
LIN {X 0,Y 510.576,Z 443.439,A -85,B 0,C 180,E1 -5411.916,E2 -5411.916} C_VEL
LIN {X 0,Y 510.931,Z 432.841,A -85,B 0,C 180,E1 -5412.815,E2 -5412.815} C_VEL
LIN {X 0,Y 511.232,Z 420.885,A -85,B 0,C 180,E1 -5413.616,E2 -5413.616} C_VEL
LIN {X 0,Y 511.339,Z 413.441,A -85,B 0,C 180,E1 -5414.019,E2 -5414.019} C_VEL
LIN {X 0,Y 509.919,Z 407.971,A -85,B 0,C 180,E1 -5414.339,E2 -5414.339} C_VEL
LIN {X 0,Y 509.883,Z 407.978,A -85,B 0,C 180,E1 -5417.652,E2 -5417.652} C_VEL
LIN {X 0,Y 509.891,Z 407.977,A -85,B 0,C 180,E1 -5420.401,E2 -5420.401} C_VEL
LIN {X 0,Y 509.826,Z 407.98,A -85,B 0,C 180,E1 -5423.564,E2 -5423.564} C_VEL
LIN {X 0,Y 509.916,Z 407.968,A -85,B 0,C 180,E1 -5426.378,E2 -5426.378} C_VEL
LIN {X 0,Y 509.881,Z 407.974,A -85,B 0,C 180,E1 -5428.844,E2 -5428.844} C_VEL
LIN {X 0,Y 509.824,Z 407.981,A -85,B 0,C 180,E1 -5431.59,E2 -5431.59} C_VEL
LIN {X 0,Y 509.851,Z 407.978,A -85,B 0,C 180,E1 -5434.414,E2 -5434.414} C_VEL
LIN {X 0,Y 509.82,Z 407.98,A -85,B 0,C 180,E1 -5437.341,E2 -5437.341} C_VEL
LIN {X 0,Y 509.841,Z 407.977,A -85,B 0,C 180,E1 -5440.382,E2 -5440.382} C_VEL
LIN {X 0,Y 509.843,Z 407.978,A -85,B 0,C 180,E1 -5443.064,E2 -5443.064} C_VEL
LIN {X 0,Y 509.833,Z 407.977,A -85,B 0,C 180,E1 -5445.792,E2 -5445.792} C_VEL
LIN {X 0,Y 509.86,Z 407.977,A -85,B 0,C 180,E1 -5448.574,E2 -5448.574} C_VEL
LIN {X 0,Y 509.869,Z 407.989,A -85,B 0,C 180,E1 -5451.221,E2 -5451.221} C_VEL
LIN {X 0,Y 511.74,Z 417.969,A -85,B 0,C 180,E1 -5453.804,E2 -5453.804} C_VEL
LIN {X 0,Y 511.399,Z 429.227,A -85,B 0,C 180,E1 -5456.417,E2 -5456.417} C_VEL
LIN {X 0,Y 511.048,Z 444.248,A -85,B 0,C 180,E1 -5459.776,E2 -5459.776} C_VEL
LIN {X 0,Y 510.77,Z 457.14,A -85,B 0,C 180,E1 -5462.551,E2 -5462.551} C_VEL
LIN {X 0,Y 510.516,Z 470.29,A -85,B 0,C 180,E1 -5465.311,E2 -5465.311} C_VEL
LIN {X 0,Y 510.299,Z 484.151,A -85,B 0,C 180,E1 -5468.17,E2 -5468.17} C_VEL
LIN {X 0,Y 510.065,Z 499.67,A -85,B 0,C 180,E1 -5471.315,E2 -5471.315} C_VEL
LIN {X 0,Y 509.882,Z 512.974,A -85,B 0,C 180,E1 -5473.998,E2 -5473.998} C_VEL
LIN {X 0,Y 509.777,Z 522.411,A -85,B 0,C 180,E1 -5475.861,E2 -5475.861} C_VEL
LIN {X 0,Y 510.845,Z 532.006,A -85,B 0,C 180,E1 -5476.078,E2 -5476.078} C_VEL
LIN {X 0,Y 511.513,Z 538.474,A -85,B 0,C 180,E1 -5476.264,E2 -5476.264} C_VEL
LIN {X 0,Y 511.192,Z 551.622,A -85,B 0,C 180,E1 -5476.737,E2 -5476.737} C_VEL
LIN {X 0,Y 510.864,Z 564.122,A -85,B 0,C 180,E1 -5477.358,E2 -5477.358} C_VEL
LIN {X 0,Y 510.586,Z 575.444,A -85,B 0,C 180,E1 -5478.084,E2 -5478.084} C_VEL
LIN {X 0,Y 510.221,Z 586.526,A -85,B 0,C 180,E1 -5478.982,E2 -5478.982} C_VEL
LIN {X 0,Y 509.947,Z 595.584,A -85,B 0,C 180,E1 -5479.879,E2 -5479.879} C_VEL
LIN {X 0,Y 509.708,Z 605.451,A -85,B 0,C 180,E1 -5481.076,E2 -5481.076} C_VEL
LIN {X 0,Y 509.513,Z 613.327,A -85,B 0,C 180,E1 -5482.271,E2 -5482.271} C_VEL
LIN {X 0,Y 509.345,Z 620.593,A -85,B 0,C 180,E1 -5483.662,E2 -5483.662} C_VEL
LIN {X 0,Y 509.276,Z 625.44,A -85,B 0,C 180,E1 -5484.853,E2 -5484.853} C_VEL
LIN {X 0,Y 509.286,Z 629.156,A -85,B 0,C 180,E1 -5486.043,E2 -5486.043} C_VEL
LIN {X 0,Y 509.231,Z 631.065,A -85,B 0,C 180,E1 -5486.835,E2 -5486.835} C_VEL
LIN {X 0,Y 509.189,Z 632.497,A -85,B 0,C 180,E1 -5487.627,E2 -5487.627} C_VEL
LIN {X 0,Y 509.089,Z 634.135,A -85,B 0,C 180,E1 -5489.209,E2 -5489.209} C_VEL
LIN {X 0,Y 509.084,Z 634.357,A -85,B 0,C 180,E1 -5490,E2 -5490} C_VEL
LIN {X 0,Y 509.089,Z 634.136,A -85,B 0,C 180,E1 -5490.791,E2 -5490.791} C_VEL
LIN {X 0,Y 509.189,Z 632.502,A -85,B 0,C 180,E1 -5492.373,E2 -5492.373} C_VEL
LIN {X 0,Y 509.231,Z 631.071,A -85,B 0,C 180,E1 -5493.164,E2 -5493.164} C_VEL
LIN {X 0,Y 509.269,Z 628.058,A -85,B 0,C 180,E1 -5494.353,E2 -5494.353} C_VEL
LIN {X 0,Y 509.344,Z 623.983,A -85,B 0,C 180,E1 -5495.543,E2 -5495.543} C_VEL
LIN {X 0,Y 509.402,Z 618.177,A -85,B 0,C 180,E1 -5496.844,E2 -5496.844} C_VEL
LIN {X 0,Y 509.563,Z 610.883,A -85,B 0,C 180,E1 -5498.127,E2 -5498.127} C_VEL
LIN {X 0,Y 509.774,Z 602.425,A -85,B 0,C 180,E1 -5499.322,E2 -5499.322} C_VEL
LIN {X 0,Y 510.031,Z 593.772,A -85,B 0,C 180,E1 -5500.319,E2 -5500.319} C_VEL
LIN {X 0,Y 510.331,Z 583.105,A -85,B 0,C 180,E1 -5501.317,E2 -5501.317} C_VEL
LIN {X 0,Y 510.618,Z 571.553,A -85,B 0,C 180,E1 -5502.187,E2 -5502.187} C_VEL
LIN {X 0,Y 510.962,Z 561.068,A -85,B 0,C 180,E1 -5502.814,E2 -5502.814} C_VEL
LIN {X 0,Y 511.203,Z 549.272,A -85,B 0,C 180,E1 -5503.364,E2 -5503.364} C_VEL
LIN {X 0,Y 511.464,Z 536.193,A -85,B 0,C 180,E1 -5503.8,E2 -5503.8} C_VEL
LIN {X 0,Y 509.872,Z 524.41,A -85,B 0,C 180,E1 -5504.098,E2 -5504.098} C_VEL
LIN {X 0,Y 509.766,Z 522.404,A -85,B 0,C 180,E1 -5504.165,E2 -5504.165} C_VEL
LIN {X 0,Y 509.987,Z 507.042,A -85,B 0,C 180,E1 -5507.235,E2 -5507.235} C_VEL
LIN {X 0,Y 510.233,Z 490.719,A -85,B 0,C 180,E1 -5510.505,E2 -5510.505} C_VEL
LIN {X 0,Y 510.453,Z 475.953,A -85,B 0,C 180,E1 -5513.533,E2 -5513.533} C_VEL
LIN {X 0,Y 510.714,Z 461.43,A -85,B 0,C 180,E1 -5516.559,E2 -5516.559} C_VEL
LIN {X 0,Y 510.977,Z 446.711,A -85,B 0,C 180,E1 -5519.679,E2 -5519.679} C_VEL
LIN {X 0,Y 511.249,Z 432.787,A -85,B 0,C 180,E1 -5522.718,E2 -5522.718} C_VEL
LIN {X 0,Y 511.681,Z 418.89,A -85,B 0,C 180,E1 -5525.867,E2 -5525.867} C_VEL
LIN {X 0,Y 511.026,Z 413.871,A -85,B 0,C 180,E1 -5527.093,E2 -5527.093} C_VEL
LIN {X 0,Y 509.887,Z 407.974,A -85,B 0,C 180,E1 -5528.65,E2 -5528.65} C_VEL
LIN {X 0,Y 509.861,Z 407.976,A -85,B 0,C 180,E1 -5531.897,E2 -5531.897} C_VEL
LIN {X 0,Y 509.858,Z 407.978,A -85,B 0,C 180,E1 -5535.332,E2 -5535.332} C_VEL
LIN {X 0,Y 509.861,Z 407.977,A -85,B 0,C 180,E1 -5538.575,E2 -5538.575} C_VEL
LIN {X 0,Y 509.853,Z 407.977,A -85,B 0,C 180,E1 -5541.786,E2 -5541.786} C_VEL
LIN {X 0,Y 509.844,Z 407.979,A -85,B 0,C 180,E1 -5544.623,E2 -5544.623} C_VEL
LIN {X 0,Y 509.862,Z 407.975,A -85,B 0,C 180,E1 -5547.481,E2 -5547.481} C_VEL
LIN {X 0,Y 509.86,Z 407.977,A -85,B 0,C 180,E1 -5550.274,E2 -5550.274} C_VEL
LIN {X 0,Y 509.89,Z 407.973,A -85,B 0,C 180,E1 -5552.945,E2 -5552.945} C_VEL
LIN {X 0,Y 509.872,Z 407.976,A -85,B 0,C 180,E1 -5555.574,E2 -5555.574} C_VEL
LIN {X 0,Y 509.824,Z 407.981,A -85,B 0,C 180,E1 -5558.149,E2 -5558.149} C_VEL
LIN {X 0,Y 509.866,Z 407.976,A -85,B 0,C 180,E1 -5560.682,E2 -5560.682} C_VEL
LIN {X 0,Y 509.887,Z 407.972,A -85,B 0,C 180,E1 -5563.175,E2 -5563.175} C_VEL
LIN {X 0,Y 509.867,Z 407.975,A -85,B 0,C 180,E1 -5565.634,E2 -5565.634} C_VEL
LIN {X 0,Y 509.924,Z 407.967,A -85,B 0,C 180,E1 -5568.875,E2 -5568.875} C_VEL
LIN {X 0,Y 509.923,Z 407.969,A -85,B 0,C 180,E1 -5572.078,E2 -5572.078} C_VEL
LIN {X 0,Y 509.985,Z 407.961,A -85,B 0,C 180,E1 -5574.464,E2 -5574.464} C_VEL
LIN {X 0,Y 510.059,Z 407.951,A -85,B 0,C 180,E1 -5577.631,E2 -5577.631} C_VEL
LIN {X 0,Y 510.068,Z 407.95,A -85,B 0,C 180,E1 -5580.79,E2 -5580.79} C_VEL
LIN {X 0,Y 509.957,Z 407.963,A -85,B 0,C 180,E1 -5583.16,E2 -5583.16} C_VEL
LIN {X 0,Y 509.98,Z 407.962,A -85,B 0,C 180,E1 -5586.33,E2 -5586.33} C_VEL
LIN {X 0,Y 509.919,Z 407.969,A -85,B 0,C 180,E1 -5588.72,E2 -5588.72} C_VEL
LIN {X 0,Y 509.907,Z 407.972,A -85,B 0,C 180,E1 -5591.932,E2 -5591.932} C_VEL
LIN {X 0,Y 509.896,Z 407.971,A -85,B 0,C 180,E1 -5595.242,E2 -5595.242} C_VEL
LIN {X 0,Y 509.891,Z 407.973,A -85,B 0,C 180,E1 -5598.001,E2 -5598.001} C_VEL
LIN {X 0,Y 509.854,Z 407.977,A -85,B 0,C 180,E1 -5601.002,E2 -5601.002} C_VEL
LIN {X 0,Y 509.84,Z 407.979,A -85,B 0,C 180,E1 -5603.563,E2 -5603.563} C_VEL
LIN {X 0,Y 509.914,Z 407.969,A -85,B 0,C 180,E1 -5606.379,E2 -5606.379} C_VEL
LIN {X 0,Y 509.879,Z 407.972,A -85,B 0,C 180,E1 -5608.844,E2 -5608.844} C_VEL
LIN {X 0,Y 509.824,Z 407.982,A -85,B 0,C 180,E1 -5611.59,E2 -5611.59} C_VEL
LIN {X 0,Y 509.855,Z 407.977,A -85,B 0,C 180,E1 -5614.413,E2 -5614.413} C_VEL
LIN {X 0,Y 509.822,Z 407.982,A -85,B 0,C 180,E1 -5617.341,E2 -5617.341} C_VEL
LIN {X 0,Y 509.841,Z 407.978,A -85,B 0,C 180,E1 -5620.382,E2 -5620.382} C_VEL
LIN {X 0,Y 509.843,Z 407.977,A -85,B 0,C 180,E1 -5623.065,E2 -5623.065} C_VEL
LIN {X 0,Y 509.834,Z 407.981,A -85,B 0,C 180,E1 -5625.793,E2 -5625.793} C_VEL
LIN {X 0,Y 509.862,Z 407.976,A -85,B 0,C 180,E1 -5628.575,E2 -5628.575} C_VEL
LIN {X 0,Y 509.855,Z 407.978,A -85,B 0,C 180,E1 -5631.787,E2 -5631.787} C_VEL
LIN {X 0,Y 509.834,Z 407.98,A -85,B 0,C 180,E1 -5633.741,E2 -5633.741} C_VEL
LIN {X 0,Y 509.168,Z 408.063,A -85,B 0,C 180,E1 -5634.4,E2 -5634.4} C_VEL
LIN {X 0,Y 506.35,Z 408.415,A -85,B 0,C 180,E1 -5635.472,E2 -5635.472} C_VEL
LIN {X 0,Y 503.958,Z 408.712,A -85,B 0,C 180,E1 -5636.336,E2 -5636.336} C_VEL
LIN {X 0,Y 502.91,Z 408.841,A -85,B 0,C 180,E1 -5637.002,E2 -5637.002} C_VEL
LIN {X 0,Y 502.813,Z 408.852,A -85,B 0,C 180,E1 -5637.228,E2 -5637.228} C_VEL
LIN {X 0,Y 502.835,Z 408.852,A -85,B 0,C 180,E1 -5640.062,E2 -5640.062} C_VEL
LIN {X 0,Y 502.838,Z 408.85,A -85,B 0,C 180,E1 -5642.534,E2 -5642.534} C_VEL
LIN {X 0,Y 502.831,Z 408.853,A -85,B 0,C 180,E1 -5645.299,E2 -5645.299} C_VEL
LIN {X 0,Y 502.785,Z 408.858,A -85,B 0,C 180,E1 -5647.827,E2 -5647.827} C_VEL
LIN {X 0,Y 502.831,Z 408.852,A -85,B 0,C 180,E1 -5650.401,E2 -5650.401} C_VEL
LIN {X 0,Y 502.838,Z 408.851,A -85,B 0,C 180,E1 -5652.932,E2 -5652.932} C_VEL
LIN {X 0,Y 502.85,Z 408.85,A -85,B 0,C 180,E1 -5655.429,E2 -5655.429} C_VEL
LIN {X 0,Y 502.883,Z 408.845,A -85,B 0,C 180,E1 -5658.717,E2 -5658.717} C_VEL
LIN {X 0,Y 502.84,Z 408.963,A -85,B 0,C 180,E1 -5659.532,E2 -5659.532} C_VEL
LIN {X 0,Y 504.478,Z 414.84,A -85,B 0,C 180,E1 -5659.87,E2 -5659.87} C_VEL
LIN {X 0,Y 504.378,Z 426.813,A -85,B 0,C 180,E1 -5660.577,E2 -5660.577} C_VEL
LIN {X 0,Y 504.004,Z 437.554,A -85,B 0,C 180,E1 -5661.379,E2 -5661.379} C_VEL
LIN {X 0,Y 503.631,Z 447.795,A -85,B 0,C 180,E1 -5662.342,E2 -5662.342} C_VEL
LIN {X 0,Y 503.369,Z 456.782,A -85,B 0,C 180,E1 -5663.386,E2 -5663.386} C_VEL
LIN {X 0,Y 503.071,Z 465.187,A -85,B 0,C 180,E1 -5664.589,E2 -5664.589} C_VEL
LIN {X 0,Y 502.865,Z 470.886,A -85,B 0,C 180,E1 -5665.592,E2 -5665.592} C_VEL
LIN {X 0,Y 502.657,Z 476.475,A -85,B 0,C 180,E1 -5666.794,E2 -5666.794} C_VEL
LIN {X 0,Y 502.537,Z 480.869,A -85,B 0,C 180,E1 -5667.997,E2 -5667.997} C_VEL
LIN {X 0,Y 502.364,Z 484.228,A -85,B 0,C 180,E1 -5669.199,E2 -5669.199} C_VEL
LIN {X 0,Y 502.313,Z 485.901,A -85,B 0,C 180,E1 -5670,E2 -5670} C_VEL
LIN {X 0,Y 502.284,Z 488.067,A -85,B 0,C 180,E1 -5671.604,E2 -5671.604} C_VEL
LIN {X 0,Y 502.271,Z 488.584,A -85,B 0,C 180,E1 -5672.406,E2 -5672.406} C_VEL
LIN {X 0,Y 502.342,Z 488.395,A -85,B 0,C 180,E1 -5674.011,E2 -5674.011} C_VEL
LIN {X 0,Y 502.354,Z 486.719,A -85,B 0,C 180,E1 -5675.62,E2 -5675.62} C_VEL
LIN {X 0,Y 502.411,Z 484.678,A -85,B 0,C 180,E1 -5676.689,E2 -5676.689} C_VEL
LIN {X 0,Y 502.475,Z 481.067,A -85,B 0,C 180,E1 -5678.04,E2 -5678.04} C_VEL
LIN {X 0,Y 502.662,Z 476.677,A -85,B 0,C 180,E1 -5679.253,E2 -5679.253} C_VEL
LIN {X 0,Y 502.896,Z 469.988,A -85,B 0,C 180,E1 -5680.671,E2 -5680.671} C_VEL
LIN {X 0,Y 503.089,Z 462.898,A -85,B 0,C 180,E1 -5681.862,E2 -5681.862} C_VEL
LIN {X 0,Y 503.373,Z 455.234,A -85,B 0,C 180,E1 -5682.908,E2 -5682.908} C_VEL
LIN {X 0,Y 503.683,Z 446.14,A -85,B 0,C 180,E1 -5683.928,E2 -5683.928} C_VEL
LIN {X 0,Y 504.006,Z 437.229,A -85,B 0,C 180,E1 -5684.743,E2 -5684.743} C_VEL
LIN {X 0,Y 504.301,Z 427.365,A -85,B 0,C 180,E1 -5685.483,E2 -5685.483} C_VEL
LIN {X 0,Y 504.584,Z 415.694,A -85,B 0,C 180,E1 -5686.175,E2 -5686.175} C_VEL
LIN {X 0,Y 502.853,Z 408.851,A -85,B 0,C 180,E1 -5686.571,E2 -5686.571} C_VEL
LIN {X 0,Y 502.829,Z 408.849,A -85,B 0,C 180,E1 -5689.6,E2 -5689.6} C_VEL
LIN {X 0,Y 502.808,Z 408.852,A -85,B 0,C 180,E1 -5692.702,E2 -5692.702} C_VEL
LIN {X 0,Y 502.827,Z 408.847,A -85,B 0,C 180,E1 -5695.677,E2 -5695.677} C_VEL
LIN {X 0,Y 502.845,Z 408.851,A -85,B 0,C 180,E1 -5698.373,E2 -5698.373} C_VEL
LIN {X 0,Y 502.798,Z 408.85,A -85,B 0,C 180,E1 -5701.499,E2 -5701.499} C_VEL
LIN {X 0,Y 502.81,Z 408.853,A -85,B 0,C 180,E1 -5704.444,E2 -5704.444} C_VEL
LIN {X 0,Y 502.786,Z 408.851,A -85,B 0,C 180,E1 -5707.178,E2 -5707.178} C_VEL
LIN {X 0,Y 502.793,Z 408.857,A -85,B 0,C 180,E1 -5710.015,E2 -5710.015} C_VEL
LIN {X 0,Y 502.808,Z 408.856,A -85,B 0,C 180,E1 -5712.199,E2 -5712.199} C_VEL
LIN {X 0,Y 502.806,Z 408.85,A -85,B 0,C 180,E1 -5715.468,E2 -5715.468} C_VEL
LIN {X 0,Y 502.825,Z 408.846,A -85,B 0,C 180,E1 -5718.934,E2 -5718.934} C_VEL
LIN {X 0,Y 502.798,Z 408.857,A -85,B 0,C 180,E1 -5722.046,E2 -5722.046} C_VEL
LIN {X 0,Y 502.804,Z 408.849,A -85,B 0,C 180,E1 -5725.034,E2 -5725.034} C_VEL
LIN {X 0,Y 502.788,Z 408.86,A -85,B 0,C 180,E1 -5727.915,E2 -5727.915} C_VEL
LIN {X 0,Y 502.829,Z 408.846,A -85,B 0,C 180,E1 -5730.712,E2 -5730.712} C_VEL
LIN {X 0,Y 502.868,Z 408.844,A -85,B 0,C 180,E1 -5733.439,E2 -5733.439} C_VEL
LIN {X 0,Y 502.78,Z 408.856,A -85,B 0,C 180,E1 -5736.085,E2 -5736.085} C_VEL
LIN {X 0,Y 502.788,Z 408.85,A -85,B 0,C 180,E1 -5738.689,E2 -5738.689} C_VEL
LIN {X 0,Y 502.831,Z 408.847,A -85,B 0,C 180,E1 -5741.248,E2 -5741.248} C_VEL
LIN {X 0,Y 502.853,Z 408.842,A -85,B 0,C 180,E1 -5744.6,E2 -5744.6} C_VEL
LIN {X 0,Y 502.865,Z 408.85,A -85,B 0,C 180,E1 -5747.627,E2 -5747.627} C_VEL
LIN {X 0,Y 504.248,Z 414.181,A -85,B 0,C 180,E1 -5747.932,E2 -5747.932} C_VEL
LIN {X 0,Y 504.218,Z 425.037,A -85,B 0,C 180,E1 -5748.568,E2 -5748.568} C_VEL
LIN {X 0,Y 503.863,Z 435.757,A -85,B 0,C 180,E1 -5749.35,E2 -5749.35} C_VEL
LIN {X 0,Y 503.517,Z 445.802,A -85,B 0,C 180,E1 -5750.256,E2 -5750.256} C_VEL
LIN {X 0,Y 503.257,Z 454.057,A -85,B 0,C 180,E1 -5751.163,E2 -5751.163} C_VEL
LIN {X 0,Y 503.005,Z 461.688,A -85,B 0,C 180,E1 -5752.17,E2 -5752.17} C_VEL
LIN {X 0,Y 502.817,Z 468.421,A -85,B 0,C 180,E1 -5753.249,E2 -5753.249} C_VEL
LIN {X 0,Y 502.608,Z 474.213,A -85,B 0,C 180,E1 -5754.383,E2 -5754.383} C_VEL
LIN {X 0,Y 502.539,Z 479.116,A -85,B 0,C 180,E1 -5755.588,E2 -5755.588} C_VEL
LIN {X 0,Y 502.409,Z 482.921,A -85,B 0,C 180,E1 -5756.792,E2 -5756.792} C_VEL
LIN {X 0,Y 502.291,Z 486.435,A -85,B 0,C 180,E1 -5758.396,E2 -5758.396} C_VEL
LIN {X 0,Y 502.239,Z 487.585,A -85,B 0,C 180,E1 -5759.198,E2 -5759.198} C_VEL
LIN {X 0,Y 502.235,Z 488.649,A -85,B 0,C 180,E1 -5760.802,E2 -5760.802} C_VEL
LIN {X 0,Y 502.279,Z 488.62,A -85,B 0,C 180,E1 -5761.603,E2 -5761.603} C_VEL
LIN {X 0,Y 502.285,Z 488.178,A -85,B 0,C 180,E1 -5762.406,E2 -5762.406} C_VEL
LIN {X 0,Y 502.384,Z 486.106,A -85,B 0,C 180,E1 -5764.011,E2 -5764.011} C_VEL
LIN {X 0,Y 502.447,Z 483.477,A -85,B 0,C 180,E1 -5765.216,E2 -5765.216} C_VEL
LIN {X 0,Y 502.58,Z 479.838,A -85,B 0,C 180,E1 -5766.423,E2 -5766.423} C_VEL
LIN {X 0,Y 502.686,Z 475.093,A -85,B 0,C 180,E1 -5767.632,E2 -5767.632} C_VEL
LIN {X 0,Y 502.915,Z 469.059,A -85,B 0,C 180,E1 -5768.842,E2 -5768.842} C_VEL
LIN {X 0,Y 503.115,Z 461.474,A -85,B 0,C 180,E1 -5770.056,E2 -5770.056} C_VEL
LIN {X 0,Y 503.439,Z 453.706,A -85,B 0,C 180,E1 -5771.067,E2 -5771.067} C_VEL
LIN {X 0,Y 503.687,Z 444.236,A -85,B 0,C 180,E1 -5772.081,E2 -5772.081} C_VEL
LIN {X 0,Y 504.052,Z 433.537,A -85,B 0,C 180,E1 -5772.993,E2 -5772.993} C_VEL
LIN {X 0,Y 504.361,Z 421.509,A -85,B 0,C 180,E1 -5773.805,E2 -5773.805} C_VEL
LIN {X 0,Y 504.489,Z 414.975,A -85,B 0,C 180,E1 -5774.162,E2 -5774.162} C_VEL
LIN {X 0,Y 502.858,Z 408.85,A -85,B 0,C 180,E1 -5774.519,E2 -5774.519} C_VEL
LIN {X 0,Y 502.825,Z 408.853,A -85,B 0,C 180,E1 -5777.069,E2 -5777.069} C_VEL
LIN {X 0,Y 502.829,Z 408.855,A -85,B 0,C 180,E1 -5779.6,E2 -5779.6} C_VEL
LIN {X 0,Y 502.807,Z 408.857,A -85,B 0,C 180,E1 -5782.702,E2 -5782.702} C_VEL
LIN {X 0,Y 502.826,Z 408.854,A -85,B 0,C 180,E1 -5785.676,E2 -5785.676} C_VEL
LIN {X 0,Y 502.844,Z 408.85,A -85,B 0,C 180,E1 -5788.372,E2 -5788.372} C_VEL
LIN {X 0,Y 502.797,Z 408.856,A -85,B 0,C 180,E1 -5791.499,E2 -5791.499} C_VEL
LIN {X 0,Y 502.807,Z 408.855,A -85,B 0,C 180,E1 -5793.994,E2 -5793.994} C_VEL
LIN {X 0,Y 502.781,Z 408.857,A -85,B 0,C 180,E1 -5797.178,E2 -5797.178} C_VEL
LIN {X 0,Y 502.791,Z 408.857,A -85,B 0,C 180,E1 -5800.015,E2 -5800.015} C_VEL
LIN {X 0,Y 502.806,Z 408.853,A -85,B 0,C 180,E1 -5802.199,E2 -5802.199} C_VEL
LIN {X 0,Y 502.804,Z 408.855,A -85,B 0,C 180,E1 -5805.468,E2 -5805.468} C_VEL
LIN {X 0,Y 502.823,Z 408.853,A -85,B 0,C 180,E1 -5808.934,E2 -5808.934} C_VEL
LIN {X 0,Y 502.808,Z 408.907,A -85,B 0,C 180,E1 -5810.96,E2 -5810.96} C_VEL
LIN {X 0,Y 504.731,Z 418.815,A -85,B 0,C 180,E1 -5813.578,E2 -5813.578} C_VEL
LIN {X 0,Y 504.736,Z 423.475,A -85,B 0,C 180,E1 -5814.7,E2 -5814.7} C_VEL
LIN {X 0,Y 504.261,Z 436.767,A -85,B 0,C 180,E1 -5817.785,E2 -5817.785} C_VEL
LIN {X 0,Y 503.907,Z 450.156,A -85,B 0,C 180,E1 -5820.781,E2 -5820.781} C_VEL
LIN {X 0,Y 503.634,Z 464.68,A -85,B 0,C 180,E1 -5823.923,E2 -5823.923} C_VEL
LIN {X 0,Y 503.333,Z 479.174,A -85,B 0,C 180,E1 -5826.985,E2 -5826.985} C_VEL
LIN {X 0,Y 503.054,Z 493.595,A -85,B 0,C 180,E1 -5829.984,E2 -5829.984} C_VEL
LIN {X 0,Y 502.871,Z 507.98,A -85,B 0,C 180,E1 -5832.933,E2 -5832.933} C_VEL
LIN {X 0,Y 502.634,Z 521.344,A -85,B 0,C 180,E1 -5835.655,E2 -5835.655} C_VEL
LIN {X 0,Y 503.958,Z 533.191,A -85,B 0,C 180,E1 -5835.939,E2 -5835.939} C_VEL
LIN {X 0,Y 504.552,Z 539.059,A -85,B 0,C 180,E1 -5836.122,E2 -5836.122} C_VEL
LIN {X 0,Y 504.214,Z 551.726,A -85,B 0,C 180,E1 -5836.601,E2 -5836.601} C_VEL
LIN {X 0,Y 503.831,Z 564.755,A -85,B 0,C 180,E1 -5837.275,E2 -5837.275} C_VEL
LIN {X 0,Y 503.535,Z 575.744,A -85,B 0,C 180,E1 -5838.017,E2 -5838.017} C_VEL
LIN {X 0,Y 503.139,Z 586.574,A -85,B 0,C 180,E1 -5838.927,E2 -5838.927} C_VEL
LIN {X 0,Y 502.866,Z 596.369,A -85,B 0,C 180,E1 -5839.939,E2 -5839.939} C_VEL
LIN {X 0,Y 502.654,Z 604.418,A -85,B 0,C 180,E1 -5840.95,E2 -5840.95} C_VEL
LIN {X 0,Y 502.428,Z 612.293,A -85,B 0,C 180,E1 -5842.161,E2 -5842.161} C_VEL
LIN {X 0,Y 502.284,Z 619.566,A -85,B 0,C 180,E1 -5843.573,E2 -5843.573} C_VEL
LIN {X 0,Y 502.236,Z 624.419,A -85,B 0,C 180,E1 -5844.781,E2 -5844.781} C_VEL
LIN {X 0,Y 502.253,Z 628.138,A -85,B 0,C 180,E1 -5845.988,E2 -5845.988} C_VEL
LIN {X 0,Y 502.187,Z 630.047,A -85,B 0,C 180,E1 -5846.791,E2 -5846.791} C_VEL
LIN {X 0,Y 502.152,Z 631.481,A -85,B 0,C 180,E1 -5847.593,E2 -5847.593} C_VEL
LIN {X 0,Y 502.086,Z 633.125,A -85,B 0,C 180,E1 -5849.198,E2 -5849.198} C_VEL
LIN {X 0,Y 502.077,Z 633.348,A -85,B 0,C 180,E1 -5850,E2 -5850} C_VEL
LIN {X 0,Y 502.086,Z 633.128,A -85,B 0,C 180,E1 -5850.802,E2 -5850.802} C_VEL
LIN {X 0,Y 502.151,Z 631.489,A -85,B 0,C 180,E1 -5852.406,E2 -5852.406} C_VEL
LIN {X 0,Y 502.187,Z 630.057,A -85,B 0,C 180,E1 -5853.209,E2 -5853.209} C_VEL
LIN {X 0,Y 502.201,Z 627.039,A -85,B 0,C 180,E1 -5854.414,E2 -5854.414} C_VEL
LIN {X 0,Y 502.285,Z 622.965,A -85,B 0,C 180,E1 -5855.621,E2 -5855.621} C_VEL
LIN {X 0,Y 502.333,Z 616.793,A -85,B 0,C 180,E1 -5857.011,E2 -5857.011} C_VEL
LIN {X 0,Y 502.494,Z 609.858,A -85,B 0,C 180,E1 -5858.242,E2 -5858.242} C_VEL
LIN {X 0,Y 502.723,Z 601.401,A -85,B 0,C 180,E1 -5859.454,E2 -5859.454} C_VEL
LIN {X 0,Y 502.968,Z 592.743,A -85,B 0,C 180,E1 -5860.466,E2 -5860.466} C_VEL
LIN {X 0,Y 503.312,Z 582.079,A -85,B 0,C 180,E1 -5861.477,E2 -5861.477} C_VEL
LIN {X 0,Y 503.589,Z 570.859,A -85,B 0,C 180,E1 -5862.336,E2 -5862.336} C_VEL
LIN {X 0,Y 503.983,Z 560.042,A -85,B 0,C 180,E1 -5862.995,E2 -5862.995} C_VEL
LIN {X 0,Y 504.312,Z 548.256,A -85,B 0,C 180,E1 -5863.55,E2 -5863.55} C_VEL
LIN {X 0,Y 504.468,Z 536.543,A -85,B 0,C 180,E1 -5863.957,E2 -5863.957} C_VEL
LIN {X 0,Y 502.938,Z 524.895,A -85,B 0,C 180,E1 -5864.271,E2 -5864.271} C_VEL
LIN {X 0,Y 502.634,Z 521.477,A -85,B 0,C 180,E1 -5864.344,E2 -5864.344} C_VEL
LIN {X 0,Y 502.931,Z 505.998,A -85,B 0,C 180,E1 -5867.484,E2 -5867.484} C_VEL
LIN {X 0,Y 503.173,Z 490.653,A -85,B 0,C 180,E1 -5870.64,E2 -5870.64} C_VEL
LIN {X 0,Y 503.436,Z 475.139,A -85,B 0,C 180,E1 -5873.881,E2 -5873.881} C_VEL
LIN {X 0,Y 503.685,Z 461.578,A -85,B 0,C 180,E1 -5876.747,E2 -5876.747} C_VEL
LIN {X 0,Y 503.967,Z 447.98,A -85,B 0,C 180,E1 -5879.674,E2 -5879.674} C_VEL
LIN {X 0,Y 504.302,Z 433.318,A -85,B 0,C 180,E1 -5882.923,E2 -5882.923} C_VEL
LIN {X 0,Y 504.725,Z 419.395,A -85,B 0,C 180,E1 -5886.136,E2 -5886.136} C_VEL
LIN {X 0,Y 503.05,Z 410.026,A -85,B 0,C 180,E1 -5888.522,E2 -5888.522} C_VEL
LIN {X 0,Y 502.823,Z 408.853,A -85,B 0,C 180,E1 -5888.84,E2 -5888.84} C_VEL
LIN {X 0,Y 502.828,Z 408.853,A -85,B 0,C 180,E1 -5891.065,E2 -5891.065} C_VEL
LIN {X 0,Y 502.802,Z 408.859,A -85,B 0,C 180,E1 -5894.532,E2 -5894.532} C_VEL
LIN {X 0,Y 502.831,Z 408.852,A -85,B 0,C 180,E1 -5897.864,E2 -5897.864} C_VEL
LIN {X 0,Y 502.804,Z 408.855,A -85,B 0,C 180,E1 -5901.024,E2 -5901.024} C_VEL
LIN {X 0,Y 502.784,Z 408.858,A -85,B 0,C 180,E1 -5904.168,E2 -5904.168} C_VEL
LIN {X 0,Y 502.834,Z 408.85,A -85,B 0,C 180,E1 -5906.993,E2 -5906.993} C_VEL
LIN {X 0,Y 502.816,Z 408.855,A -85,B 0,C 180,E1 -5910.065,E2 -5910.065} C_VEL
LIN {X 0,Y 502.838,Z 408.851,A -85,B 0,C 180,E1 -5912.533,E2 -5912.533} C_VEL
LIN {X 0,Y 502.831,Z 408.852,A -85,B 0,C 180,E1 -5915.298,E2 -5915.298} C_VEL
LIN {X 0,Y 502.787,Z 408.858,A -85,B 0,C 180,E1 -5917.827,E2 -5917.827} C_VEL
LIN {X 0,Y 502.827,Z 408.853,A -85,B 0,C 180,E1 -5920.4,E2 -5920.4} C_VEL
LIN {X 0,Y 502.837,Z 408.851,A -85,B 0,C 180,E1 -5922.932,E2 -5922.932} C_VEL
LIN {X 0,Y 502.847,Z 408.85,A -85,B 0,C 180,E1 -5925.429,E2 -5925.429} C_VEL
LIN {X 0,Y 502.894,Z 408.843,A -85,B 0,C 180,E1 -5928.717,E2 -5928.717} C_VEL
LIN {X 0,Y 502.883,Z 408.846,A -85,B 0,C 180,E1 -5931.966,E2 -5931.966} C_VEL
LIN {X 0,Y 502.941,Z 408.839,A -85,B 0,C 180,E1 -5934.387,E2 -5934.387} C_VEL
LIN {X 0,Y 503.029,Z 408.827,A -85,B 0,C 180,E1 -5937.598,E2 -5937.598} C_VEL
LIN {X 0,Y 503.029,Z 408.828,A -85,B 0,C 180,E1 -5940,E2 -5940} C_VEL
LIN {X 0,Y 503.025,Z 408.828,A -85,B 0,C 180,E1 -5942.402,E2 -5942.402} C_VEL
LIN {X 0,Y 502.94,Z 408.839,A -85,B 0,C 180,E1 -5945.614,E2 -5945.614} C_VEL
LIN {X 0,Y 502.905,Z 408.844,A -85,B 0,C 180,E1 -5948.033,E2 -5948.033} C_VEL
LIN {X 0,Y 502.88,Z 408.846,A -85,B 0,C 180,E1 -5951.283,E2 -5951.283} C_VEL
LIN {X 0,Y 502.848,Z 408.849,A -85,B 0,C 180,E1 -5954.571,E2 -5954.571} C_VEL
LIN {X 0,Y 502.864,Z 408.848,A -85,B 0,C 180,E1 -5957.907,E2 -5957.907} C_VEL
LIN {X 0,Y 502.832,Z 408.853,A -85,B 0,C 180,E1 -5960.537,E2 -5960.537} C_VEL
LIN {X 0,Y 502.8,Z 408.855,A -85,B 0,C 180,E1 -5963.04,E2 -5963.04} C_VEL
LIN {X 0,Y 502.843,Z 408.851,A -85,B 0,C 180,E1 -5965.676,E2 -5965.676} C_VEL
LIN {X 0,Y 502.843,Z 408.851,A -85,B 0,C 180,E1 -5968.373,E2 -5968.373} C_VEL
LIN {X 0,Y 502.796,Z 408.857,A -85,B 0,C 180,E1 -5971.499,E2 -5971.499} C_VEL
LIN {X 0,Y 502.808,Z 408.855,A -85,B 0,C 180,E1 -5974.445,E2 -5974.445} C_VEL
LIN {X 0,Y 502.784,Z 408.858,A -85,B 0,C 180,E1 -5977.179,E2 -5977.179} C_VEL
LIN {X 0,Y 502.79,Z 408.858,A -85,B 0,C 180,E1 -5980.015,E2 -5980.015} C_VEL
LIN {X 0,Y 502.805,Z 408.856,A -85,B 0,C 180,E1 -5982.199,E2 -5982.199} C_VEL
LIN {X 0,Y 502.804,Z 408.855,A -85,B 0,C 180,E1 -5985.468,E2 -5985.468} C_VEL
LIN {X 0,Y 502.833,Z 408.854,A -85,B 0,C 180,E1 -5987.865,E2 -5987.865} C_VEL
LIN {X 0,Y 502.805,Z 408.854,A -85,B 0,C 180,E1 -5991.024,E2 -5991.024} C_VEL
LIN {X 0,Y 502.788,Z 408.859,A -85,B 0,C 180,E1 -5994.168,E2 -5994.168} C_VEL
LIN {X 0,Y 502.813,Z 408.852,A -85,B 0,C 180,E1 -5997.228,E2 -5997.228} C_VEL
LIN {X 0,Y 502.116,Z 408.942,A -85,B 0,C 180,E1 -5997.896,E2 -5997.896} C_VEL
LIN {X 0,Y 499.258,Z 409.297,A -85,B 0,C 180,E1 -5998.982,E2 -5998.982} C_VEL
LIN {X 0,Y 496.865,Z 409.597,A -85,B 0,C 180,E1 -5999.857,E2 -5999.857} C_VEL
LIN {X 0,Y 495.847,Z 409.721,A -85,B 0,C 180,E1 -6000.533,E2 -6000.533} C_VEL
LIN {X 0,Y 495.768,Z 409.73,A -85,B 0,C 180,E1 -6000.762,E2 -6000.762} C_VEL
LIN {X 0,Y 495.795,Z 409.73,A -85,B 0,C 180,E1 -6003.932,E2 -6003.932} C_VEL
LIN {X 0,Y 495.764,Z 409.731,A -85,B 0,C 180,E1 -6007.139,E2 -6007.139} C_VEL
LIN {X 0,Y 495.783,Z 409.73,A -85,B 0,C 180,E1 -6010.11,E2 -6010.11} C_VEL
LIN {X 0,Y 495.791,Z 409.728,A -85,B 0,C 180,E1 -6012.682,E2 -6012.682} C_VEL
LIN {X 0,Y 495.795,Z 409.729,A -85,B 0,C 180,E1 -6015.217,E2 -6015.217} C_VEL
LIN {X 0,Y 495.857,Z 409.721,A -85,B 0,C 180,E1 -6018.555,E2 -6018.555} C_VEL
LIN {X 0,Y 495.806,Z 409.861,A -85,B 0,C 180,E1 -6019.33,E2 -6019.33} C_VEL
LIN {X 0,Y 497.709,Z 416.65,A -85,B 0,C 180,E1 -6019.731,E2 -6019.731} C_VEL
LIN {X 0,Y 497.52,Z 428.472,A -85,B 0,C 180,E1 -6020.446,E2 -6020.446} C_VEL
LIN {X 0,Y 497.128,Z 439.045,A -85,B 0,C 180,E1 -6021.259,E2 -6021.259} C_VEL
LIN {X 0,Y 496.719,Z 449.204,A -85,B 0,C 180,E1 -6022.234,E2 -6022.234} C_VEL
LIN {X 0,Y 496.427,Z 458.125,A -85,B 0,C 180,E1 -6023.293,E2 -6023.293} C_VEL
LIN {X 0,Y 496.118,Z 466.448,A -85,B 0,C 180,E1 -6024.513,E2 -6024.513} C_VEL
LIN {X 0,Y 495.886,Z 472.119,A -85,B 0,C 180,E1 -6025.529,E2 -6025.529} C_VEL
LIN {X 0,Y 495.672,Z 477.653,A -85,B 0,C 180,E1 -6026.749,E2 -6026.749} C_VEL
LIN {X 0,Y 495.549,Z 482.006,A -85,B 0,C 180,E1 -6027.968,E2 -6027.968} C_VEL
LIN {X 0,Y 495.364,Z 485.334,A -85,B 0,C 180,E1 -6029.187,E2 -6029.187} C_VEL
LIN {X 0,Y 495.226,Z 488.248,A -85,B 0,C 180,E1 -6030.813,E2 -6030.813} C_VEL
LIN {X 0,Y 495.273,Z 489.118,A -85,B 0,C 180,E1 -6031.626,E2 -6031.626} C_VEL
LIN {X 0,Y 495.245,Z 489.608,A -85,B 0,C 180,E1 -6032.44,E2 -6032.44} C_VEL
LIN {X 0,Y 495.315,Z 489.383,A -85,B 0,C 180,E1 -6034.068,E2 -6034.068} C_VEL
LIN {X 0,Y 495.338,Z 488.718,A -85,B 0,C 180,E1 -6034.884,E2 -6034.884} C_VEL
LIN {X 0,Y 495.347,Z 487.661,A -85,B 0,C 180,E1 -6035.7,E2 -6035.7} C_VEL
LIN {X 0,Y 495.457,Z 484.266,A -85,B 0,C 180,E1 -6037.335,E2 -6037.335} C_VEL
LIN {X 0,Y 495.573,Z 480.571,A -85,B 0,C 180,E1 -6038.564,E2 -6038.564} C_VEL
LIN {X 0,Y 495.768,Z 475.756,A -85,B 0,C 180,E1 -6039.795,E2 -6039.795} C_VEL
LIN {X 0,Y 496.013,Z 469.674,A -85,B 0,C 180,E1 -6041.028,E2 -6041.028} C_VEL
LIN {X 0,Y 496.262,Z 462.043,A -85,B 0,C 180,E1 -6042.265,E2 -6042.265} C_VEL
LIN {X 0,Y 496.578,Z 454.2,A -85,B 0,C 180,E1 -6043.296,E2 -6043.296} C_VEL
LIN {X 0,Y 496.882,Z 444.594,A -85,B 0,C 180,E1 -6044.331,E2 -6044.331} C_VEL
LIN {X 0,Y 497.319,Z 433.842,A -85,B 0,C 180,E1 -6045.261,E2 -6045.261} C_VEL
LIN {X 0,Y 497.64,Z 423.228,A -85,B 0,C 180,E1 -6045.988,E2 -6045.988} C_VEL
LIN {X 0,Y 497.791,Z 417.642,A -85,B 0,C 180,E1 -6046.307,E2 -6046.307} C_VEL
LIN {X 0,Y 495.796,Z 409.729,A -85,B 0,C 180,E1 -6046.788,E2 -6046.788} C_VEL
LIN {X 0,Y 495.776,Z 409.729,A -85,B 0,C 180,E1 -6049.89,E2 -6049.89} C_VEL
LIN {X 0,Y 495.764,Z 409.728,A -85,B 0,C 180,E1 -6052.861,E2 -6052.861} C_VEL
LIN {X 0,Y 495.786,Z 409.728,A -85,B 0,C 180,E1 -6056.068,E2 -6056.068} C_VEL
LIN {X 0,Y 495.776,Z 409.726,A -85,B 0,C 180,E1 -6058.815,E2 -6058.815} C_VEL
LIN {X 0,Y 495.76,Z 409.728,A -85,B 0,C 180,E1 -6061.725,E2 -6061.725} C_VEL
LIN {X 0,Y 495.78,Z 409.726,A -85,B 0,C 180,E1 -6064.695,E2 -6064.695} C_VEL
LIN {X 0,Y 495.736,Z 409.73,A -85,B 0,C 180,E1 -6067.561,E2 -6067.561} C_VEL
LIN {X 0,Y 495.771,Z 409.726,A -85,B 0,C 180,E1 -6070.7,E2 -6070.7} C_VEL
LIN {X 0,Y 495.739,Z 409.736,A -85,B 0,C 180,E1 -6074.001,E2 -6074.001} C_VEL
LIN {X 0,Y 495.731,Z 409.73,A -85,B 0,C 180,E1 -6077.117,E2 -6077.117} C_VEL
LIN {X 0,Y 495.763,Z 409.734,A -85,B 0,C 180,E1 -6079.953,E2 -6079.953} C_VEL
LIN {X 0,Y 495.732,Z 409.731,A -85,B 0,C 180,E1 -6082.553,E2 -6082.553} C_VEL
LIN {X 0,Y 495.782,Z 409.726,A -85,B 0,C 180,E1 -6085.457,E2 -6085.457} C_VEL
LIN {X 0,Y 495.76,Z 409.729,A -85,B 0,C 180,E1 -6088.364,E2 -6088.364} C_VEL
LIN {X 0,Y 495.792,Z 409.726,A -85,B 0,C 180,E1 -6091.507,E2 -6091.507} C_VEL
LIN {X 0,Y 495.786,Z 409.73,A -85,B 0,C 180,E1 -6093.932,E2 -6093.932} C_VEL
LIN {X 0,Y 495.764,Z 409.727,A -85,B 0,C 180,E1 -6097.139,E2 -6097.139} C_VEL
LIN {X 0,Y 495.776,Z 409.728,A -85,B 0,C 180,E1 -6100.11,E2 -6100.11} C_VEL
LIN {X 0,Y 495.768,Z 409.725,A -85,B 0,C 180,E1 -6102.681,E2 -6102.681} C_VEL
LIN {X 0,Y 495.795,Z 409.724,A -85,B 0,C 180,E1 -6105.217,E2 -6105.217} C_VEL
LIN {X 0,Y 495.814,Z 409.727,A -85,B 0,C 180,E1 -6107.443,E2 -6107.443} C_VEL
LIN {X 0,Y 497.483,Z 416.698,A -85,B 0,C 180,E1 -6107.855,E2 -6107.855} C_VEL
LIN {X 0,Y 497.224,Z 427.315,A -85,B 0,C 180,E1 -6108.5,E2 -6108.5} C_VEL
LIN {X 0,Y 496.878,Z 437.883,A -85,B 0,C 180,E1 -6109.301,E2 -6109.301} C_VEL
LIN {X 0,Y 496.596,Z 447.716,A -85,B 0,C 180,E1 -6110.222,E2 -6110.222} C_VEL
LIN {X 0,Y 496.244,Z 456.603,A -85,B 0,C 180,E1 -6111.243,E2 -6111.243} C_VEL
LIN {X 0,Y 495.978,Z 465.26,A -85,B 0,C 180,E1 -6112.468,E2 -6112.468} C_VEL
LIN {X 0,Y 495.819,Z 472.221,A -85,B 0,C 180,E1 -6113.693,E2 -6113.693} C_VEL
LIN {X 0,Y 495.54,Z 476.935,A -85,B 0,C 180,E1 -6114.71,E2 -6114.71} C_VEL
LIN {X 0,Y 495.447,Z 481.488,A -85,B 0,C 180,E1 -6115.933,E2 -6115.933} C_VEL
LIN {X 0,Y 495.389,Z 483.902,A -85,B 0,C 180,E1 -6116.747,E2 -6116.747} C_VEL
LIN {X 0,Y 495.281,Z 487.433,A -85,B 0,C 180,E1 -6118.374,E2 -6118.374} C_VEL
LIN {X 0,Y 495.223,Z 488.584,A -85,B 0,C 180,E1 -6119.187,E2 -6119.187} C_VEL
LIN {X 0,Y 495.219,Z 489.656,A -85,B 0,C 180,E1 -6120.813,E2 -6120.813} C_VEL
LIN {X 0,Y 495.269,Z 489.63,A -85,B 0,C 180,E1 -6121.626,E2 -6121.626} C_VEL
LIN {X 0,Y 495.262,Z 489.184,A -85,B 0,C 180,E1 -6122.44,E2 -6122.44} C_VEL
LIN {X 0,Y 495.368,Z 487.113,A -85,B 0,C 180,E1 -6124.068,E2 -6124.068} C_VEL
LIN {X 0,Y 495.456,Z 484.471,A -85,B 0,C 180,E1 -6125.29,E2 -6125.29} C_VEL
LIN {X 0,Y 495.599,Z 480.818,A -85,B 0,C 180,E1 -6126.514,E2 -6126.514} C_VEL
LIN {X 0,Y 495.721,Z 476.053,A -85,B 0,C 180,E1 -6127.74,E2 -6127.74} C_VEL
LIN {X 0,Y 495.97,Z 469.977,A -85,B 0,C 180,E1 -6128.967,E2 -6128.967} C_VEL
LIN {X 0,Y 496.195,Z 462.359,A -85,B 0,C 180,E1 -6130.198,E2 -6130.198} C_VEL
LIN {X 0,Y 496.524,Z 454.553,A -85,B 0,C 180,E1 -6131.223,E2 -6131.223} C_VEL
LIN {X 0,Y 496.79,Z 445.022,A -85,B 0,C 180,E1 -6132.251,E2 -6132.251} C_VEL
LIN {X 0,Y 497.186,Z 434.241,A -85,B 0,C 180,E1 -6133.176,E2 -6133.176} C_VEL
LIN {X 0,Y 497.509,Z 423.785,A -85,B 0,C 180,E1 -6133.895,E2 -6133.895} C_VEL
LIN {X 0,Y 497.643,Z 416.539,A -85,B 0,C 180,E1 -6134.309,E2 -6134.309} C_VEL
LIN {X 0,Y 495.837,Z 409.725,A -85,B 0,C 180,E1 -6134.703,E2 -6134.703} C_VEL
LIN {X 0,Y 495.785,Z 409.732,A -85,B 0,C 180,E1 -6138.171,E2 -6138.171} C_VEL
LIN {X 0,Y 495.778,Z 409.733,A -85,B 0,C 180,E1 -6140.756,E2 -6140.756} C_VEL
LIN {X 0,Y 495.747,Z 409.735,A -85,B 0,C 180,E1 -6143.387,E2 -6143.387} C_VEL
LIN {X 0,Y 495.828,Z 409.723,A -85,B 0,C 180,E1 -6146.749,E2 -6146.749} C_VEL
LIN {X 0,Y 495.77,Z 409.731,A -85,B 0,C 180,E1 -6149.746,E2 -6149.746} C_VEL
LIN {X 0,Y 495.771,Z 409.732,A -85,B 0,C 180,E1 -6152.594,E2 -6152.594} C_VEL
LIN {X 0,Y 495.751,Z 409.734,A -85,B 0,C 180,E1 -6155.537,E2 -6155.537} C_VEL
LIN {X 0,Y 495.766,Z 409.73,A -85,B 0,C 180,E1 -6158.768,E2 -6158.768} C_VEL
LIN {X 0,Y 495.781,Z 409.726,A -85,B 0,C 180,E1 -6161.779,E2 -6161.779} C_VEL
LIN {X 0,Y 495.753,Z 409.736,A -85,B 0,C 180,E1 -6165.139,E2 -6165.139} C_VEL
LIN {X 0,Y 495.76,Z 409.733,A -85,B 0,C 180,E1 -6168.219,E2 -6168.219} C_VEL
LIN {X 0,Y 495.793,Z 409.827,A -85,B 0,C 180,E1 -6170.702,E2 -6170.702} C_VEL
LIN {X 0,Y 497.586,Z 418.745,A -85,B 0,C 180,E1 -6173.11,E2 -6173.11} C_VEL
LIN {X 0,Y 497.94,Z 422.854,A -85,B 0,C 180,E1 -6174.145,E2 -6174.145} C_VEL
LIN {X 0,Y 497.305,Z 437.108,A -85,B 0,C 180,E1 -6177.519,E2 -6177.519} C_VEL
LIN {X 0,Y 496.956,Z 449.416,A -85,B 0,C 180,E1 -6180.332,E2 -6180.332} C_VEL
LIN {X 0,Y 496.666,Z 462.86,A -85,B 0,C 180,E1 -6183.303,E2 -6183.303} C_VEL
LIN {X 0,Y 496.313,Z 478.348,A -85,B 0,C 180,E1 -6186.641,E2 -6186.641} C_VEL
LIN {X 0,Y 496.043,Z 491.704,A -85,B 0,C 180,E1 -6189.472,E2 -6189.472} C_VEL
LIN {X 0,Y 495.804,Z 507.044,A -85,B 0,C 180,E1 -6192.682,E2 -6192.682} C_VEL
LIN {X 0,Y 495.582,Z 520.29,A -85,B 0,C 180,E1 -6195.447,E2 -6195.447} C_VEL
LIN {X 0,Y 496.901,Z 533.06,A -85,B 0,C 180,E1 -6195.761,E2 -6195.761} C_VEL
LIN {X 0,Y 497.594,Z 539.56,A -85,B 0,C 180,E1 -6195.977,E2 -6195.977} C_VEL
LIN {X 0,Y 497.181,Z 552.962,A -85,B 0,C 180,E1 -6196.512,E2 -6196.512} C_VEL
LIN {X 0,Y 496.769,Z 565.635,A -85,B 0,C 180,E1 -6197.215,E2 -6197.215} C_VEL
LIN {X 0,Y 496.454,Z 577.332,A -85,B 0,C 180,E1 -6198.051,E2 -6198.051} C_VEL
LIN {X 0,Y 496.068,Z 587.698,A -85,B 0,C 180,E1 -6198.973,E2 -6198.973} C_VEL
LIN {X 0,Y 495.765,Z 597.05,A -85,B 0,C 180,E1 -6199.999,E2 -6199.999} C_VEL
LIN {X 0,Y 495.495,Z 606.182,A -85,B 0,C 180,E1 -6201.229,E2 -6201.229} C_VEL
LIN {X 0,Y 495.32,Z 613.554,A -85,B 0,C 180,E1 -6202.458,E2 -6202.458} C_VEL
LIN {X 0,Y 495.228,Z 619.457,A -85,B 0,C 180,E1 -6203.686,E2 -6203.686} C_VEL
LIN {X 0,Y 495.169,Z 624.747,A -85,B 0,C 180,E1 -6205.115,E2 -6205.115} C_VEL
LIN {X 0,Y 495.215,Z 627.119,A -85,B 0,C 180,E1 -6205.931,E2 -6205.931} C_VEL
LIN {X 0,Y 495.145,Z 629.029,A -85,B 0,C 180,E1 -6206.745,E2 -6206.745} C_VEL
LIN {X 0,Y 495.114,Z 630.465,A -85,B 0,C 180,E1 -6207.559,E2 -6207.559} C_VEL
LIN {X 0,Y 495.08,Z 632.116,A -85,B 0,C 180,E1 -6209.186,E2 -6209.186} C_VEL
LIN {X 0,Y 495.069,Z 632.339,A -85,B 0,C 180,E1 -6210,E2 -6210} C_VEL
LIN {X 0,Y 495.08,Z 632.119,A -85,B 0,C 180,E1 -6210.813,E2 -6210.813} C_VEL
LIN {X 0,Y 495.113,Z 630.476,A -85,B 0,C 180,E1 -6212.44,E2 -6212.44} C_VEL
LIN {X 0,Y 495.144,Z 629.043,A -85,B 0,C 180,E1 -6213.255,E2 -6213.255} C_VEL
LIN {X 0,Y 495.144,Z 626.023,A -85,B 0,C 180,E1 -6214.477,E2 -6214.477} C_VEL
LIN {X 0,Y 495.266,Z 620.744,A -85,B 0,C 180,E1 -6216.003,E2 -6216.003} C_VEL
LIN {X 0,Y 495.277,Z 614.631,A -85,B 0,C 180,E1 -6217.337,E2 -6217.337} C_VEL
LIN {X 0,Y 495.47,Z 607.572,A -85,B 0,C 180,E1 -6218.565,E2 -6218.565} C_VEL
LIN {X 0,Y 495.684,Z 598.747,A -85,B 0,C 180,E1 -6219.796,E2 -6219.796} C_VEL
LIN {X 0,Y 496.002,Z 589.733,A -85,B 0,C 180,E1 -6220.821,E2 -6220.821} C_VEL
LIN {X 0,Y 496.373,Z 579.865,A -85,B 0,C 180,E1 -6221.743,E2 -6221.743} C_VEL
LIN {X 0,Y 496.638,Z 569.672,A -85,B 0,C 180,E1 -6222.524,E2 -6222.524} C_VEL
LIN {X 0,Y 497.052,Z 557.064,A -85,B 0,C 180,E1 -6223.283,E2 -6223.283} C_VEL
LIN {X 0,Y 497.417,Z 544.608,A -85,B 0,C 180,E1 -6223.846,E2 -6223.846} C_VEL
LIN {X 0,Y 497.436,Z 536.866,A -85,B 0,C 180,E1 -6224.119,E2 -6224.119} C_VEL
LIN {X 0,Y 496.033,Z 525.359,A -85,B 0,C 180,E1 -6224.448,E2 -6224.448} C_VEL
LIN {X 0,Y 495.569,Z 520.304,A -85,B 0,C 180,E1 -6224.579,E2 -6224.579} C_VEL
LIN {X 0,Y 495.849,Z 506.121,A -85,B 0,C 180,E1 -6227.529,E2 -6227.529} C_VEL
LIN {X 0,Y 496.102,Z 490.627,A -85,B 0,C 180,E1 -6230.774,E2 -6230.774} C_VEL
LIN {X 0,Y 496.386,Z 475.32,A -85,B 0,C 180,E1 -6234.02,E2 -6234.02} C_VEL
LIN {X 0,Y 496.664,Z 460.843,A -85,B 0,C 180,E1 -6237.129,E2 -6237.129} C_VEL
LIN {X 0,Y 496.945,Z 449.233,A -85,B 0,C 180,E1 -6239.669,E2 -6239.669} C_VEL
LIN {X 0,Y 497.305,Z 435.644,A -85,B 0,C 180,E1 -6242.721,E2 -6242.721} C_VEL
LIN {X 0,Y 497.79,Z 422.148,A -85,B 0,C 180,E1 -6245.867,E2 -6245.867} C_VEL
LIN {X 0,Y 497.37,Z 417.972,A -85,B 0,C 180,E1 -6246.908,E2 -6246.908} C_VEL
LIN {X 0,Y 495.801,Z 409.728,A -85,B 0,C 180,E1 -6249.114,E2 -6249.114} C_VEL
LIN {X 0,Y 495.761,Z 409.733,A -85,B 0,C 180,E1 -6251.781,E2 -6251.781} C_VEL
LIN {X 0,Y 495.751,Z 409.736,A -85,B 0,C 180,E1 -6255.139,E2 -6255.139} C_VEL
LIN {X 0,Y 495.779,Z 409.731,A -85,B 0,C 180,E1 -6258.221,E2 -6258.221} C_VEL
LIN {X 0,Y 495.753,Z 409.733,A -85,B 0,C 180,E1 -6261.409,E2 -6261.409} C_VEL
LIN {X 0,Y 495.757,Z 409.735,A -85,B 0,C 180,E1 -6264.463,E2 -6264.463} C_VEL
LIN {X 0,Y 495.769,Z 409.73,A -85,B 0,C 180,E1 -6267.406,E2 -6267.406} C_VEL
LIN {X 0,Y 495.768,Z 409.732,A -85,B 0,C 180,E1 -6270.254,E2 -6270.254} C_VEL
LIN {X 0,Y 495.836,Z 409.723,A -85,B 0,C 180,E1 -6273.248,E2 -6273.248} C_VEL
LIN {X 0,Y 495.755,Z 409.734,A -85,B 0,C 180,E1 -6275.725,E2 -6275.725} C_VEL
LIN {X 0,Y 495.746,Z 409.736,A -85,B 0,C 180,E1 -6278.371,E2 -6278.371} C_VEL
LIN {X 0,Y 495.786,Z 409.728,A -85,B 0,C 180,E1 -6280.972,E2 -6280.972} C_VEL
LIN {X 0,Y 495.782,Z 409.729,A -85,B 0,C 180,E1 -6283.53,E2 -6283.53} C_VEL
LIN {X 0,Y 495.797,Z 409.73,A -85,B 0,C 180,E1 -6286.056,E2 -6286.056} C_VEL
LIN {X 0,Y 495.87,Z 409.719,A -85,B 0,C 180,E1 -6288.555,E2 -6288.555} C_VEL
LIN {X 0,Y 495.839,Z 409.724,A -85,B 0,C 180,E1 -6291.852,E2 -6291.852} C_VEL
LIN {X 0,Y 495.899,Z 409.716,A -85,B 0,C 180,E1 -6294.307,E2 -6294.307} C_VEL
LIN {X 0,Y 495.998,Z 409.703,A -85,B 0,C 180,E1 -6297.564,E2 -6297.564} C_VEL
LIN {X 0,Y 496,Z 409.704,A -85,B 0,C 180,E1 -6300,E2 -6300} C_VEL
LIN {X 0,Y 495.994,Z 409.704,A -85,B 0,C 180,E1 -6302.436,E2 -6302.436} C_VEL
LIN {X 0,Y 495.898,Z 409.717,A -85,B 0,C 180,E1 -6305.694,E2 -6305.694} C_VEL
LIN {X 0,Y 495.876,Z 409.719,A -85,B 0,C 180,E1 -6308.148,E2 -6308.148} C_VEL
LIN {X 0,Y 495.854,Z 409.721,A -85,B 0,C 180,E1 -6311.445,E2 -6311.445} C_VEL
LIN {X 0,Y 495.793,Z 409.727,A -85,B 0,C 180,E1 -6314.783,E2 -6314.783} C_VEL
LIN {X 0,Y 495.789,Z 409.728,A -85,B 0,C 180,E1 -6317.319,E2 -6317.319} C_VEL
LIN {X 0,Y 495.781,Z 409.732,A -85,B 0,C 180,E1 -6319.89,E2 -6319.89} C_VEL
LIN {X 0,Y 495.761,Z 409.732,A -85,B 0,C 180,E1 -6322.861,E2 -6322.861} C_VEL
LIN {X 0,Y 495.794,Z 409.73,A -85,B 0,C 180,E1 -6326.068,E2 -6326.068} C_VEL
LIN {X 0,Y 495.774,Z 409.729,A -85,B 0,C 180,E1 -6328.815,E2 -6328.815} C_VEL
LIN {X 0,Y 495.759,Z 409.735,A -85,B 0,C 180,E1 -6331.726,E2 -6331.726} C_VEL
LIN {X 0,Y 495.778,Z 409.73,A -85,B 0,C 180,E1 -6334.695,E2 -6334.695} C_VEL
LIN {X 0,Y 495.734,Z 409.736,A -85,B 0,C 180,E1 -6337.562,E2 -6337.562} C_VEL
LIN {X 0,Y 495.769,Z 409.729,A -85,B 0,C 180,E1 -6340.7,E2 -6340.7} C_VEL
LIN {X 0,Y 495.738,Z 409.737,A -85,B 0,C 180,E1 -6343.696,E2 -6343.696} C_VEL
LIN {X 0,Y 495.738,Z 409.735,A -85,B 0,C 180,E1 -6346.305,E2 -6346.305} C_VEL
LIN {X 0,Y 495.77,Z 409.732,A -85,B 0,C 180,E1 -6349.301,E2 -6349.301} C_VEL
LIN {X 0,Y 495.734,Z 409.734,A -85,B 0,C 180,E1 -6352.439,E2 -6352.439} C_VEL
LIN {X 0,Y 495.788,Z 409.73,A -85,B 0,C 180,E1 -6355.458,E2 -6355.458} C_VEL
LIN {X 0,Y 495.764,Z 409.733,A -85,B 0,C 180,E1 -6358.364,E2 -6358.364} C_VEL
LIN {X 0,Y 495.768,Z 409.73,A -85,B 0,C 180,E1 -6360.762,E2 -6360.762} C_VEL
LIN {X 0,Y 495.106,Z 409.815,A -85,B 0,C 180,E1 -6361.441,E2 -6361.441} C_VEL
LIN {X 0,Y 492.245,Z 410.169,A -85,B 0,C 180,E1 -6362.543,E2 -6362.543} C_VEL
LIN {X 0,Y 489.835,Z 410.471,A -85,B 0,C 180,E1 -6363.431,E2 -6363.431} C_VEL
LIN {X 0,Y 488.819,Z 410.598,A -85,B 0,C 180,E1 -6364.118,E2 -6364.118} C_VEL
LIN {X 0,Y 488.747,Z 410.604,A -85,B 0,C 180,E1 -6364.35,E2 -6364.35} C_VEL
LIN {X 0,Y 488.727,Z 410.608,A -85,B 0,C 180,E1 -6367.153,E2 -6367.153} C_VEL
LIN {X 0,Y 488.734,Z 410.609,A -85,B 0,C 180,E1 -6369.811,E2 -6369.811} C_VEL
LIN {X 0,Y 488.739,Z 410.607,A -85,B 0,C 180,E1 -6372.424,E2 -6372.424} C_VEL
LIN {X 0,Y 488.767,Z 410.605,A -85,B 0,C 180,E1 -6375,E2 -6375} C_VEL
LIN {X 0,Y 488.811,Z 410.599,A -85,B 0,C 180,E1 -6378.388,E2 -6378.388} C_VEL
LIN {X 0,Y 488.789,Z 410.74,A -85,B 0,C 180,E1 -6379.122,E2 -6379.122} C_VEL
LIN {X 0,Y 490.908,Z 418.467,A -85,B 0,C 180,E1 -6379.587,E2 -6379.587} C_VEL
LIN {X 0,Y 490.65,Z 430.111,A -85,B 0,C 180,E1 -6380.311,E2 -6380.311} C_VEL
LIN {X 0,Y 490.245,Z 440.535,A -85,B 0,C 180,E1 -6381.135,E2 -6381.135} C_VEL
LIN {X 0,Y 489.818,Z 450.611,A -85,B 0,C 180,E1 -6382.124,E2 -6382.124} C_VEL
LIN {X 0,Y 489.491,Z 459.468,A -85,B 0,C 180,E1 -6383.197,E2 -6383.197} C_VEL
LIN {X 0,Y 489.162,Z 467.708,A -85,B 0,C 180,E1 -6384.435,E2 -6384.435} C_VEL
LIN {X 0,Y 488.907,Z 473.344,A -85,B 0,C 180,E1 -6385.466,E2 -6385.466} C_VEL
LIN {X 0,Y 488.685,Z 478.826,A -85,B 0,C 180,E1 -6386.702,E2 -6386.702} C_VEL
LIN {X 0,Y 488.559,Z 483.14,A -85,B 0,C 180,E1 -6387.939,E2 -6387.939} C_VEL
LIN {X 0,Y 488.362,Z 486.435,A -85,B 0,C 180,E1 -6389.176,E2 -6389.176} C_VEL
LIN {X 0,Y 488.208,Z 489.315,A -85,B 0,C 180,E1 -6390.825,E2 -6390.825} C_VEL
LIN {X 0,Y 488.261,Z 490.168,A -85,B 0,C 180,E1 -6391.65,E2 -6391.65} C_VEL
LIN {X 0,Y 488.219,Z 490.628,A -85,B 0,C 180,E1 -6392.475,E2 -6392.475} C_VEL
LIN {X 0,Y 488.29,Z 490.371,A -85,B 0,C 180,E1 -6394.127,E2 -6394.127} C_VEL
LIN {X 0,Y 488.332,Z 489.688,A -85,B 0,C 180,E1 -6394.954,E2 -6394.954} C_VEL
LIN {X 0,Y 488.341,Z 488.599,A -85,B 0,C 180,E1 -6395.782,E2 -6395.782} C_VEL
LIN {X 0,Y 488.473,Z 485.168,A -85,B 0,C 180,E1 -6397.44,E2 -6397.44} C_VEL
LIN {X 0,Y 488.605,Z 481.436,A -85,B 0,C 180,E1 -6398.687,E2 -6398.687} C_VEL
LIN {X 0,Y 488.822,Z 476.581,A -85,B 0,C 180,E1 -6399.935,E2 -6399.935} C_VEL
LIN {X 0,Y 489.071,Z 470.456,A -85,B 0,C 180,E1 -6401.186,E2 -6401.186} C_VEL
LIN {X 0,Y 489.344,Z 462.748,A -85,B 0,C 180,E1 -6402.441,E2 -6402.441} C_VEL
LIN {X 0,Y 489.676,Z 454.843,A -85,B 0,C 180,E1 -6403.487,E2 -6403.487} C_VEL
LIN {X 0,Y 489.998,Z 445.162,A -85,B 0,C 180,E1 -6404.537,E2 -6404.537} C_VEL
LIN {X 0,Y 490.483,Z 434.271,A -85,B 0,C 180,E1 -6405.479,E2 -6405.479} C_VEL
LIN {X 0,Y 490.823,Z 423.499,A -85,B 0,C 180,E1 -6406.216,E2 -6406.216} C_VEL
LIN {X 0,Y 490.832,Z 418.142,A -85,B 0,C 180,E1 -6406.528,E2 -6406.528} C_VEL
LIN {X 0,Y 488.767,Z 410.603,A -85,B 0,C 180,E1 -6406.982,E2 -6406.982} C_VEL
LIN {X 0,Y 488.73,Z 410.609,A -85,B 0,C 180,E1 -6410.19,E2 -6410.19} C_VEL
LIN {X 0,Y 488.714,Z 410.605,A -85,B 0,C 180,E1 -6413.02,E2 -6413.02} C_VEL
LIN {X 0,Y 488.732,Z 410.602,A -85,B 0,C 180,E1 -6415.557,E2 -6415.557} C_VEL
LIN {X 0,Y 488.749,Z 410.607,A -85,B 0,C 180,E1 -6418.329,E2 -6418.329} C_VEL
LIN {X 0,Y 488.697,Z 410.606,A -85,B 0,C 180,E1 -6421.18,E2 -6421.18} C_VEL
LIN {X 0,Y 488.739,Z 410.608,A -85,B 0,C 180,E1 -6424.113,E2 -6424.113} C_VEL
LIN {X 0,Y 488.687,Z 410.607,A -85,B 0,C 180,E1 -6427.159,E2 -6427.159} C_VEL
LIN {X 0,Y 488.723,Z 410.608,A -85,B 0,C 180,E1 -6430.345,E2 -6430.345} C_VEL
LIN {X 0,Y 488.691,Z 410.609,A -85,B 0,C 180,E1 -6433.654,E2 -6433.654} C_VEL
LIN {X 0,Y 488.692,Z 410.611,A -85,B 0,C 180,E1 -6436.346,E2 -6436.346} C_VEL
LIN {X 0,Y 488.738,Z 410.605,A -85,B 0,C 180,E1 -6439.677,E2 -6439.677} C_VEL
LIN {X 0,Y 488.684,Z 410.608,A -85,B 0,C 180,E1 -6442.841,E2 -6442.841} C_VEL
LIN {X 0,Y 488.735,Z 410.609,A -85,B 0,C 180,E1 -6445.887,E2 -6445.887} C_VEL
LIN {X 0,Y 488.697,Z 410.606,A -85,B 0,C 180,E1 -6448.82,E2 -6448.82} C_VEL
LIN {X 0,Y 488.749,Z 410.605,A -85,B 0,C 180,E1 -6451.671,E2 -6451.671} C_VEL
LIN {X 0,Y 488.732,Z 410.603,A -85,B 0,C 180,E1 -6454.443,E2 -6454.443} C_VEL
LIN {X 0,Y 488.726,Z 410.603,A -85,B 0,C 180,E1 -6457.153,E2 -6457.153} C_VEL
LIN {X 0,Y 488.73,Z 410.61,A -85,B 0,C 180,E1 -6459.81,E2 -6459.81} C_VEL
LIN {X 0,Y 488.719,Z 410.604,A -85,B 0,C 180,E1 -6462.423,E2 -6462.423} C_VEL
LIN {X 0,Y 488.767,Z 410.598,A -85,B 0,C 180,E1 -6465,E2 -6465} C_VEL
LIN {X 0,Y 488.794,Z 410.6,A -85,B 0,C 180,E1 -6467.26,E2 -6467.26} C_VEL
LIN {X 0,Y 490.562,Z 417.601,A -85,B 0,C 180,E1 -6467.681,E2 -6467.681} C_VEL
LIN {X 0,Y 490.325,Z 428.282,A -85,B 0,C 180,E1 -6468.342,E2 -6468.342} C_VEL
LIN {X 0,Y 489.946,Z 439.997,A -85,B 0,C 180,E1 -6469.253,E2 -6469.253} C_VEL
LIN {X 0,Y 489.663,Z 448.614,A -85,B 0,C 180,E1 -6470.082,E2 -6470.082} C_VEL
LIN {X 0,Y 489.3,Z 457.513,A -85,B 0,C 180,E1 -6471.117,E2 -6471.117} C_VEL
LIN {X 0,Y 489.011,Z 466.191,A -85,B 0,C 180,E1 -6472.36,E2 -6472.36} C_VEL
LIN {X 0,Y 488.837,Z 473.167,A -85,B 0,C 180,E1 -6473.603,E2 -6473.603} C_VEL
LIN {X 0,Y 488.546,Z 477.897,A -85,B 0,C 180,E1 -6474.635,E2 -6474.635} C_VEL
LIN {X 0,Y 488.434,Z 482.465,A -85,B 0,C 180,E1 -6475.874,E2 -6475.874} C_VEL
LIN {X 0,Y 488.369,Z 484.883,A -85,B 0,C 180,E1 -6476.7,E2 -6476.7} C_VEL
LIN {X 0,Y 488.27,Z 488.432,A -85,B 0,C 180,E1 -6478.35,E2 -6478.35} C_VEL
LIN {X 0,Y 488.206,Z 489.583,A -85,B 0,C 180,E1 -6479.175,E2 -6479.175} C_VEL
LIN {X 0,Y 488.202,Z 490.668,A -85,B 0,C 180,E1 -6480.825,E2 -6480.825} C_VEL
LIN {X 0,Y 488.258,Z 490.64,A -85,B 0,C 180,E1 -6481.65,E2 -6481.65} C_VEL
LIN {X 0,Y 488.298,Z 489.344,A -85,B 0,C 180,E1 -6483.3,E2 -6483.3} C_VEL
LIN {X 0,Y 488.353,Z 488.119,A -85,B 0,C 180,E1 -6484.126,E2 -6484.126} C_VEL
LIN {X 0,Y 488.466,Z 485.466,A -85,B 0,C 180,E1 -6485.366,E2 -6485.366} C_VEL
LIN {X 0,Y 488.62,Z 481.797,A -85,B 0,C 180,E1 -6486.607,E2 -6486.607} C_VEL
LIN {X 0,Y 488.755,Z 477.01,A -85,B 0,C 180,E1 -6487.851,E2 -6487.851} C_VEL
LIN {X 0,Y 489.026,Z 470.895,A -85,B 0,C 180,E1 -6489.096,E2 -6489.096} C_VEL
LIN {X 0,Y 489.281,Z 463.257,A -85,B 0,C 180,E1 -6490.343,E2 -6490.343} C_VEL
LIN {X 0,Y 489.612,Z 455.43,A -85,B 0,C 180,E1 -6491.383,E2 -6491.383} C_VEL
LIN {X 0,Y 489.901,Z 445.85,A -85,B 0,C 180,E1 -6492.426,E2 -6492.426} C_VEL
LIN {X 0,Y 490.337,Z 435.028,A -85,B 0,C 180,E1 -6493.363,E2 -6493.363} C_VEL
LIN {X 0,Y 490.667,Z 424.526,A -85,B 0,C 180,E1 -6494.093,E2 -6494.093} C_VEL
LIN {X 0,Y 490.558,Z 417.208,A -85,B 0,C 180,E1 -6494.52,E2 -6494.52} C_VEL
LIN {X 0,Y 488.78,Z 410.603,A -85,B 0,C 180,E1 -6494.92,E2 -6494.92} C_VEL
LIN {X 0,Y 488.751,Z 410.61,A -85,B 0,C 180,E1 -6498.442,E2 -6498.442} C_VEL
LIN {X 0,Y 488.711,Z 410.613,A -85,B 0,C 180,E1 -6501.071,E2 -6501.071} C_VEL
LIN {X 0,Y 488.684,Z 410.614,A -85,B 0,C 180,E1 -6503.746,E2 -6503.746} C_VEL
LIN {X 0,Y 488.796,Z 410.6,A -85,B 0,C 180,E1 -6506.944,E2 -6506.944} C_VEL
LIN {X 0,Y 488.713,Z 410.61,A -85,B 0,C 180,E1 -6510.363,E2 -6510.363} C_VEL
LIN {X 0,Y 488.738,Z 410.605,A -85,B 0,C 180,E1 -6513.484,E2 -6513.484} C_VEL
LIN {X 0,Y 488.685,Z 410.613,A -85,B 0,C 180,E1 -6516.354,E2 -6516.354} C_VEL
LIN {X 0,Y 488.704,Z 410.61,A -85,B 0,C 180,E1 -6519.254,E2 -6519.254} C_VEL
LIN {X 0,Y 488.726,Z 410.605,A -85,B 0,C 180,E1 -6521.602,E2 -6521.602} C_VEL
LIN {X 0,Y 488.716,Z 410.61,A -85,B 0,C 180,E1 -6524.801,E2 -6524.801} C_VEL
LIN {X 0,Y 488.695,Z 410.612,A -85,B 0,C 180,E1 -6527.474,E2 -6527.474} C_VEL
LIN {X 0,Y 488.748,Z 410.693,A -85,B 0,C 180,E1 -6530.417,E2 -6530.417} C_VEL
LIN {X 0,Y 490.818,Z 421.254,A -85,B 0,C 180,E1 -6533.308,E2 -6533.308} C_VEL
LIN {X 0,Y 490.915,Z 425.74,A -85,B 0,C 180,E1 -6534.434,E2 -6534.434} C_VEL
LIN {X 0,Y 490.306,Z 439.55,A -85,B 0,C 180,E1 -6537.747,E2 -6537.747} C_VEL
LIN {X 0,Y 489.923,Z 451.771,A -85,B 0,C 180,E1 -6540.572,E2 -6540.572} C_VEL
LIN {X 0,Y 489.57,Z 465.171,A -85,B 0,C 180,E1 -6543.575,E2 -6543.575} C_VEL
LIN {X 0,Y 489.222,Z 480.078,A -85,B 0,C 180,E1 -6546.839,E2 -6546.839} C_VEL
LIN {X 0,Y 488.958,Z 492.204,A -85,B 0,C 180,E1 -6549.455,E2 -6549.455} C_VEL
LIN {X 0,Y 488.73,Z 507.118,A -85,B 0,C 180,E1 -6552.639,E2 -6552.639} C_VEL
LIN {X 0,Y 488.513,Z 519.256,A -85,B 0,C 180,E1 -6555.231,E2 -6555.231} C_VEL
LIN {X 0,Y 489.795,Z 532.92,A -85,B 0,C 180,E1 -6555.576,E2 -6555.576} C_VEL
LIN {X 0,Y 490.629,Z 540.059,A -85,B 0,C 180,E1 -6555.826,E2 -6555.826} C_VEL
LIN {X 0,Y 490.193,Z 552.964,A -85,B 0,C 180,E1 -6556.369,E2 -6556.369} C_VEL
LIN {X 0,Y 489.772,Z 565.296,A -85,B 0,C 180,E1 -6557.075,E2 -6557.075} C_VEL
LIN {X 0,Y 489.422,Z 576.29,A -85,B 0,C 180,E1 -6557.877,E2 -6557.877} C_VEL
LIN {X 0,Y 488.976,Z 586.651,A -85,B 0,C 180,E1 -6558.811,E2 -6558.811} C_VEL
LIN {X 0,Y 488.714,Z 596.013,A -85,B 0,C 180,E1 -6559.853,E2 -6559.853} C_VEL
LIN {X 0,Y 488.436,Z 605.148,A -85,B 0,C 180,E1 -6561.102,E2 -6561.102} C_VEL
LIN {X 0,Y 488.266,Z 612.524,A -85,B 0,C 180,E1 -6562.349,E2 -6562.349} C_VEL
LIN {X 0,Y 488.165,Z 618.767,A -85,B 0,C 180,E1 -6563.678,E2 -6563.678} C_VEL
LIN {X 0,Y 488.121,Z 623.725,A -85,B 0,C 180,E1 -6565.044,E2 -6565.044} C_VEL
LIN {X 0,Y 488.157,Z 626.098,A -85,B 0,C 180,E1 -6565.872,E2 -6565.872} C_VEL
LIN {X 0,Y 488.102,Z 628.011,A -85,B 0,C 180,E1 -6566.698,E2 -6566.698} C_VEL
LIN {X 0,Y 488.075,Z 629.449,A -85,B 0,C 180,E1 -6567.524,E2 -6567.524} C_VEL
LIN {X 0,Y 488.072,Z 631.106,A -85,B 0,C 180,E1 -6569.175,E2 -6569.175} C_VEL
LIN {X 0,Y 488.06,Z 631.329,A -85,B 0,C 180,E1 -6570,E2 -6570} C_VEL
LIN {X 0,Y 488.072,Z 631.11,A -85,B 0,C 180,E1 -6570.825,E2 -6570.825} C_VEL
LIN {X 0,Y 488.074,Z 629.463,A -85,B 0,C 180,E1 -6572.476,E2 -6572.476} C_VEL
LIN {X 0,Y 488.1,Z 628.029,A -85,B 0,C 180,E1 -6573.302,E2 -6573.302} C_VEL
LIN {X 0,Y 488.094,Z 625.007,A -85,B 0,C 180,E1 -6574.542,E2 -6574.542} C_VEL
LIN {X 0,Y 488.203,Z 619.896,A -85,B 0,C 180,E1 -6576.048,E2 -6576.048} C_VEL
LIN {X 0,Y 488.239,Z 613.612,A -85,B 0,C 180,E1 -6577.444,E2 -6577.444} C_VEL
LIN {X 0,Y 488.402,Z 606.547,A -85,B 0,C 180,E1 -6578.69,E2 -6578.69} C_VEL
LIN {X 0,Y 488.634,Z 597.721,A -85,B 0,C 180,E1 -6579.939,E2 -6579.939} C_VEL
LIN {X 0,Y 488.989,Z 587.71,A -85,B 0,C 180,E1 -6581.083,E2 -6581.083} C_VEL
LIN {X 0,Y 489.405,Z 577.661,A -85,B 0,C 180,E1 -6582.017,E2 -6582.017} C_VEL
LIN {X 0,Y 489.739,Z 567.129,A -85,B 0,C 180,E1 -6582.81,E2 -6582.81} C_VEL
LIN {X 0,Y 490.114,Z 555.033,A -85,B 0,C 180,E1 -6583.527,E2 -6583.527} C_VEL
LIN {X 0,Y 490.557,Z 542.279,A -85,B 0,C 180,E1 -6584.096,E2 -6584.096} C_VEL
LIN {X 0,Y 490.386,Z 537.008,A -85,B 0,C 180,E1 -6584.286,E2 -6584.286} C_VEL
LIN {X 0,Y 489.094,Z 525.532,A -85,B 0,C 180,E1 -6584.631,E2 -6584.631} C_VEL
LIN {X 0,Y 488.514,Z 519.387,A -85,B 0,C 180,E1 -6584.768,E2 -6584.768} C_VEL
LIN {X 0,Y 488.776,Z 504.293,A -85,B 0,C 180,E1 -6587.98,E2 -6587.98} C_VEL
LIN {X 0,Y 489.054,Z 488.876,A -85,B 0,C 180,E1 -6591.276,E2 -6591.276} C_VEL
LIN {X 0,Y 489.371,Z 474.438,A -85,B 0,C 180,E1 -6594.386,E2 -6594.386} C_VEL
LIN {X 0,Y 489.654,Z 460.906,A -85,B 0,C 180,E1 -6597.342,E2 -6597.342} C_VEL
LIN {X 0,Y 489.963,Z 449.426,A -85,B 0,C 180,E1 -6599.898,E2 -6599.898} C_VEL
LIN {X 0,Y 490.359,Z 435.866,A -85,B 0,C 180,E1 -6602.999,E2 -6602.999} C_VEL
LIN {X 0,Y 490.856,Z 423.435,A -85,B 0,C 180,E1 -6605.947,E2 -6605.947} C_VEL
LIN {X 0,Y 490.085,Z 417.589,A -85,B 0,C 180,E1 -6607.442,E2 -6607.442} C_VEL
LIN {X 0,Y 488.761,Z 410.604,A -85,B 0,C 180,E1 -6609.315,E2 -6609.315} C_VEL
LIN {X 0,Y 488.693,Z 410.614,A -85,B 0,C 180,E1 -6612.525,E2 -6612.525} C_VEL
LIN {X 0,Y 488.713,Z 410.612,A -85,B 0,C 180,E1 -6615.199,E2 -6615.199} C_VEL
LIN {X 0,Y 488.725,Z 410.609,A -85,B 0,C 180,E1 -6618.398,E2 -6618.398} C_VEL
LIN {X 0,Y 488.706,Z 410.611,A -85,B 0,C 180,E1 -6620.947,E2 -6620.947} C_VEL
LIN {X 0,Y 488.685,Z 410.614,A -85,B 0,C 180,E1 -6623.868,E2 -6623.868} C_VEL
LIN {X 0,Y 488.74,Z 410.606,A -85,B 0,C 180,E1 -6626.877,E2 -6626.877} C_VEL
LIN {X 0,Y 488.725,Z 410.609,A -85,B 0,C 180,E1 -6629.781,E2 -6629.781} C_VEL
LIN {X 0,Y 488.801,Z 410.599,A -85,B 0,C 180,E1 -6633.055,E2 -6633.055} C_VEL
LIN {X 0,Y 488.696,Z 410.614,A -85,B 0,C 180,E1 -6636.255,E2 -6636.255} C_VEL
LIN {X 0,Y 488.747,Z 410.604,A -85,B 0,C 180,E1 -6639.176,E2 -6639.176} C_VEL
LIN {X 0,Y 488.761,Z 410.604,A -85,B 0,C 180,E1 -6641.628,E2 -6641.628} C_VEL
LIN {X 0,Y 488.764,Z 410.603,A -85,B 0,C 180,E1 -6645,E2 -6645} C_VEL
LIN {X 0,Y 488.832,Z 410.596,A -85,B 0,C 180,E1 -6648.388,E2 -6648.388} C_VEL
LIN {X 0,Y 488.788,Z 410.603,A -85,B 0,C 180,E1 -6651.733,E2 -6651.733} C_VEL
LIN {X 0,Y 488.858,Z 410.593,A -85,B 0,C 180,E1 -6654.224,E2 -6654.224} C_VEL
LIN {X 0,Y 488.965,Z 410.579,A -85,B 0,C 180,E1 -6657.529,E2 -6657.529} C_VEL
LIN {X 0,Y 488.958,Z 410.579,A -85,B 0,C 180,E1 -6660.824,E2 -6660.824} C_VEL
LIN {X 0,Y 488.962,Z 410.579,A -85,B 0,C 180,E1 -6662.471,E2 -6662.471} C_VEL
LIN {X 0,Y 488.857,Z 410.594,A -85,B 0,C 180,E1 -6665.776,E2 -6665.776} C_VEL
LIN {X 0,Y 488.82,Z 410.597,A -85,B 0,C 180,E1 -6668.267,E2 -6668.267} C_VEL
LIN {X 0,Y 488.808,Z 410.599,A -85,B 0,C 180,E1 -6671.613,E2 -6671.613} C_VEL
LIN {X 0,Y 488.765,Z 410.602,A -85,B 0,C 180,E1 -6675.001,E2 -6675.001} C_VEL
LIN {X 0,Y 488.757,Z 410.606,A -85,B 0,C 180,E1 -6678.442,E2 -6678.442} C_VEL
LIN {X 0,Y 488.711,Z 410.61,A -85,B 0,C 180,E1 -6681.071,E2 -6681.071} C_VEL
LIN {X 0,Y 488.697,Z 410.613,A -85,B 0,C 180,E1 -6683.746,E2 -6683.746} C_VEL
LIN {X 0,Y 488.794,Z 410.599,A -85,B 0,C 180,E1 -6686.944,E2 -6686.944} C_VEL
LIN {X 0,Y 488.712,Z 410.612,A -85,B 0,C 180,E1 -6690.363,E2 -6690.363} C_VEL
LIN {X 0,Y 488.738,Z 410.607,A -85,B 0,C 180,E1 -6693.485,E2 -6693.485} C_VEL
LIN {X 0,Y 488.691,Z 410.613,A -85,B 0,C 180,E1 -6696.356,E2 -6696.356} C_VEL
LIN {X 0,Y 488.703,Z 410.612,A -85,B 0,C 180,E1 -6699.254,E2 -6699.254} C_VEL
LIN {X 0,Y 488.726,Z 410.61,A -85,B 0,C 180,E1 -6701.602,E2 -6701.602} C_VEL
LIN {X 0,Y 488.715,Z 410.609,A -85,B 0,C 180,E1 -6704.802,E2 -6704.802} C_VEL
LIN {X 0,Y 488.698,Z 410.612,A -85,B 0,C 180,E1 -6707.475,E2 -6707.475} C_VEL
LIN {X 0,Y 488.736,Z 410.608,A -85,B 0,C 180,E1 -6709.677,E2 -6709.677} C_VEL
LIN {X 0,Y 488.685,Z 410.612,A -85,B 0,C 180,E1 -6712.842,E2 -6712.842} C_VEL
LIN {X 0,Y 488.738,Z 410.608,A -85,B 0,C 180,E1 -6715.888,E2 -6715.888} C_VEL
LIN {X 0,Y 488.701,Z 410.611,A -85,B 0,C 180,E1 -6718.821,E2 -6718.821} C_VEL
LIN {X 0,Y 488.75,Z 410.607,A -85,B 0,C 180,E1 -6721.672,E2 -6721.672} C_VEL
LIN {X 0,Y 488.747,Z 410.604,A -85,B 0,C 180,E1 -6724.35,E2 -6724.35} C_VEL
LIN {X 0,Y 488.102,Z 410.687,A -85,B 0,C 180,E1 -6725.038,E2 -6725.038} C_VEL
LIN {X 0,Y 485.234,Z 411.047,A -85,B 0,C 180,E1 -6726.154,E2 -6726.154} C_VEL
LIN {X 0,Y 482.787,Z 411.351,A -85,B 0,C 180,E1 -6727.054,E2 -6727.054} C_VEL
LIN {X 0,Y 481.729,Z 411.481,A -85,B 0,C 180,E1 -6727.749,E2 -6727.749} C_VEL
LIN {X 0,Y 481.64,Z 411.49,A -85,B 0,C 180,E1 -6727.985,E2 -6727.985} C_VEL
LIN {X 0,Y 481.713,Z 411.482,A -85,B 0,C 180,E1 -6730.393,E2 -6730.393} C_VEL
LIN {X 0,Y 481.695,Z 411.485,A -85,B 0,C 180,E1 -6733.034,E2 -6733.034} C_VEL
LIN {X 0,Y 481.694,Z 411.485,A -85,B 0,C 180,E1 -6735.639,E2 -6735.639} C_VEL
LIN {X 0,Y 481.779,Z 411.519,A -85,B 0,C 180,E1 -6738.909,E2 -6738.909} C_VEL
LIN {X 0,Y 484.068,Z 420.236,A -85,B 0,C 180,E1 -6739.438,E2 -6739.438} C_VEL
LIN {X 0,Y 483.781,Z 431.675,A -85,B 0,C 180,E1 -6740.172,E2 -6740.172} C_VEL
LIN {X 0,Y 483.328,Z 442.234,A -85,B 0,C 180,E1 -6741.028,E2 -6741.028} C_VEL
LIN {X 0,Y 482.879,Z 452.771,A -85,B 0,C 180,E1 -6742.095,E2 -6742.095} C_VEL
LIN {X 0,Y 482.558,Z 460.801,A -85,B 0,C 180,E1 -6743.099,E2 -6743.099} C_VEL
LIN {X 0,Y 482.207,Z 468.965,A -85,B 0,C 180,E1 -6744.354,E2 -6744.354} C_VEL
LIN {X 0,Y 481.929,Z 474.558,A -85,B 0,C 180,E1 -6745.4,E2 -6745.4} C_VEL
LIN {X 0,Y 481.697,Z 479.999,A -85,B 0,C 180,E1 -6746.654,E2 -6746.654} C_VEL
LIN {X 0,Y 481.566,Z 484.274,A -85,B 0,C 180,E1 -6747.909,E2 -6747.909} C_VEL
LIN {X 0,Y 481.358,Z 487.534,A -85,B 0,C 180,E1 -6749.164,E2 -6749.164} C_VEL
LIN {X 0,Y 481.303,Z 489.147,A -85,B 0,C 180,E1 -6750,E2 -6750} C_VEL
LIN {X 0,Y 481.19,Z 490.383,A -85,B 0,C 180,E1 -6750.837,E2 -6750.837} C_VEL
LIN {X 0,Y 481.248,Z 491.216,A -85,B 0,C 180,E1 -6751.674,E2 -6751.674} C_VEL
LIN {X 0,Y 481.232,Z 491.687,A -85,B 0,C 180,E1 -6753.349,E2 -6753.349} C_VEL
LIN {X 0,Y 481.327,Z 490.657,A -85,B 0,C 180,E1 -6755.026,E2 -6755.026} C_VEL
LIN {X 0,Y 481.335,Z 489.537,A -85,B 0,C 180,E1 -6755.867,E2 -6755.867} C_VEL
LIN {X 0,Y 481.43,Z 487.535,A -85,B 0,C 180,E1 -6756.935,E2 -6756.935} C_VEL
LIN {X 0,Y 481.545,Z 483.696,A -85,B 0,C 180,E1 -6758.392,E2 -6758.392} C_VEL
LIN {X 0,Y 481.784,Z 479.18,A -85,B 0,C 180,E1 -6759.658,E2 -6759.658} C_VEL
LIN {X 0,Y 482.088,Z 472.337,A -85,B 0,C 180,E1 -6761.138,E2 -6761.138} C_VEL
LIN {X 0,Y 482.359,Z 465.508,A -85,B 0,C 180,E1 -6762.313,E2 -6762.313} C_VEL
LIN {X 0,Y 482.739,Z 457.253,A -85,B 0,C 180,E1 -6763.47,E2 -6763.47} C_VEL
LIN {X 0,Y 483.118,Z 446.811,A -85,B 0,C 180,E1 -6764.641,E2 -6764.641} C_VEL
LIN {X 0,Y 483.61,Z 436.113,A -85,B 0,C 180,E1 -6765.596,E2 -6765.596} C_VEL
LIN {X 0,Y 483.949,Z 425.876,A -85,B 0,C 180,E1 -6766.327,E2 -6766.327} C_VEL
LIN {X 0,Y 484.123,Z 420.661,A -85,B 0,C 180,E1 -6766.639,E2 -6766.639} C_VEL
LIN {X 0,Y 481.707,Z 411.482,A -85,B 0,C 180,E1 -6767.212,E2 -6767.212} C_VEL
LIN {X 0,Y 481.71,Z 411.48,A -85,B 0,C 180,E1 -6769.607,E2 -6769.607} C_VEL
LIN {X 0,Y 481.654,Z 411.491,A -85,B 0,C 180,E1 -6772.295,E2 -6772.295} C_VEL
LIN {X 0,Y 481.694,Z 411.478,A -85,B 0,C 180,E1 -6775.231,E2 -6775.231} C_VEL
LIN {X 0,Y 481.705,Z 411.48,A -85,B 0,C 180,E1 -6777.832,E2 -6777.832} C_VEL
LIN {X 0,Y 481.65,Z 411.486,A -85,B 0,C 180,E1 -6780.711,E2 -6780.711} C_VEL
LIN {X 0,Y 481.702,Z 411.48,A -85,B 0,C 180,E1 -6783.733,E2 -6783.733} C_VEL
LIN {X 0,Y 481.633,Z 411.487,A -85,B 0,C 180,E1 -6786.747,E2 -6786.747} C_VEL
LIN {X 0,Y 481.681,Z 411.486,A -85,B 0,C 180,E1 -6789.94,E2 -6789.94} C_VEL
LIN {X 0,Y 481.644,Z 411.485,A -85,B 0,C 180,E1 -6793.3,E2 -6793.3} C_VEL
LIN {X 0,Y 481.663,Z 411.485,A -85,B 0,C 180,E1 -6795.641,E2 -6795.641} C_VEL
LIN {X 0,Y 481.661,Z 411.482,A -85,B 0,C 180,E1 -6798.958,E2 -6798.958} C_VEL
LIN {X 0,Y 481.659,Z 411.491,A -85,B 0,C 180,E1 -6801.993,E2 -6801.993} C_VEL
LIN {X 0,Y 481.693,Z 411.48,A -85,B 0,C 180,E1 -6805.318,E2 -6805.318} C_VEL
LIN {X 0,Y 481.649,Z 411.487,A -85,B 0,C 180,E1 -6808.312,E2 -6808.312} C_VEL
LIN {X 0,Y 481.704,Z 411.478,A -85,B 0,C 180,E1 -6811.219,E2 -6811.219} C_VEL
LIN {X 0,Y 481.694,Z 411.484,A -85,B 0,C 180,E1 -6814.042,E2 -6814.042} C_VEL
LIN {X 0,Y 481.679,Z 411.48,A -85,B 0,C 180,E1 -6816.812,E2 -6816.812} C_VEL
LIN {X 0,Y 481.7,Z 411.482,A -85,B 0,C 180,E1 -6819.503,E2 -6819.503} C_VEL
LIN {X 0,Y 481.696,Z 411.481,A -85,B 0,C 180,E1 -6822.158,E2 -6822.158} C_VEL
LIN {X 0,Y 481.747,Z 411.472,A -85,B 0,C 180,E1 -6824.776,E2 -6824.776} C_VEL
LIN {X 0,Y 481.744,Z 411.477,A -85,B 0,C 180,E1 -6827.07,E2 -6827.07} C_VEL
LIN {X 0,Y 483.716,Z 419.043,A -85,B 0,C 180,E1 -6827.536,E2 -6827.536} C_VEL
LIN {X 0,Y 483.326,Z 430.352,A -85,B 0,C 180,E1 -6828.254,E2 -6828.254} C_VEL
LIN {X 0,Y 483.038,Z 440.886,A -85,B 0,C 180,E1 -6829.097,E2 -6829.097} C_VEL
LIN {X 0,Y 482.735,Z 449.513,A -85,B 0,C 180,E1 -6829.938,E2 -6829.938} C_VEL
LIN {X 0,Y 482.359,Z 458.426,A -85,B 0,C 180,E1 -6830.989,E2 -6830.989} C_VEL
LIN {X 0,Y 482.047,Z 467.123,A -85,B 0,C 180,E1 -6832.249,E2 -6832.249} C_VEL
LIN {X 0,Y 481.854,Z 474.113,A -85,B 0,C 180,E1 -6833.509,E2 -6833.509} C_VEL
LIN {X 0,Y 481.48,Z 480.499,A -85,B 0,C 180,E1 -6834.975,E2 -6834.975} C_VEL
LIN {X 0,Y 481.497,Z 484.682,A -85,B 0,C 180,E1 -6836.234,E2 -6836.234} C_VEL
LIN {X 0,Y 481.242,Z 487.858,A -85,B 0,C 180,E1 -6837.489,E2 -6837.489} C_VEL
LIN {X 0,Y 481.257,Z 489.431,A -85,B 0,C 180,E1 -6838.326,E2 -6838.326} C_VEL
LIN {X 0,Y 481.188,Z 490.582,A -85,B 0,C 180,E1 -6839.163,E2 -6839.163} C_VEL
LIN {X 0,Y 481.185,Z 491.68,A -85,B 0,C 180,E1 -6840.837,E2 -6840.837} C_VEL
LIN {X 0,Y 481.246,Z 491.65,A -85,B 0,C 180,E1 -6841.674,E2 -6841.674} C_VEL
LIN {X 0,Y 481.28,Z 490.356,A -85,B 0,C 180,E1 -6843.348,E2 -6843.348} C_VEL
LIN {X 0,Y 481.339,Z 489.13,A -85,B 0,C 180,E1 -6844.186,E2 -6844.186} C_VEL
LIN {X 0,Y 481.474,Z 486.469,A -85,B 0,C 180,E1 -6845.444,E2 -6845.444} C_VEL
LIN {X 0,Y 481.642,Z 482.794,A -85,B 0,C 180,E1 -6846.704,E2 -6846.704} C_VEL
LIN {X 0,Y 481.793,Z 477.994,A -85,B 0,C 180,E1 -6847.965,E2 -6847.965} C_VEL
LIN {X 0,Y 482.084,Z 471.86,A -85,B 0,C 180,E1 -6849.228,E2 -6849.228} C_VEL
LIN {X 0,Y 482.371,Z 464.199,A -85,B 0,C 180,E1 -6850.493,E2 -6850.493} C_VEL
LIN {X 0,Y 482.707,Z 456.344,A -85,B 0,C 180,E1 -6851.548,E2 -6851.548} C_VEL
LIN {X 0,Y 483.02,Z 446.7,A -85,B 0,C 180,E1 -6852.606,E2 -6852.606} C_VEL
LIN {X 0,Y 483.489,Z 435.834,A -85,B 0,C 180,E1 -6853.556,E2 -6853.556} C_VEL
LIN {X 0,Y 483.837,Z 425.273,A -85,B 0,C 180,E1 -6854.296,E2 -6854.296} C_VEL
LIN {X 0,Y 483.915,Z 419.871,A -85,B 0,C 180,E1 -6854.616,E2 -6854.616} C_VEL
LIN {X 0,Y 481.738,Z 411.48,A -85,B 0,C 180,E1 -6855.143,E2 -6855.143} C_VEL
LIN {X 0,Y 481.713,Z 411.488,A -85,B 0,C 180,E1 -6858.722,E2 -6858.722} C_VEL
LIN {X 0,Y 481.65,Z 411.494,A -85,B 0,C 180,E1 -6861.395,E2 -6861.395} C_VEL
LIN {X 0,Y 481.665,Z 411.49,A -85,B 0,C 180,E1 -6864.114,E2 -6864.114} C_VEL
LIN {X 0,Y 481.751,Z 411.48,A -85,B 0,C 180,E1 -6867.139,E2 -6867.139} C_VEL
LIN {X 0,Y 481.683,Z 411.486,A -85,B 0,C 180,E1 -6869.741,E2 -6869.741} C_VEL
LIN {X 0,Y 481.675,Z 411.489,A -85,B 0,C 180,E1 -6872.674,E2 -6872.674} C_VEL
LIN {X 0,Y 481.64,Z 411.492,A -85,B 0,C 180,E1 -6875.709,E2 -6875.709} C_VEL
LIN {X 0,Y 481.674,Z 411.486,A -85,B 0,C 180,E1 -6878.859,E2 -6878.859} C_VEL
LIN {X 0,Y 481.668,Z 411.485,A -85,B 0,C 180,E1 -6882.159,E2 -6882.159} C_VEL
LIN {X 0,Y 481.663,Z 411.488,A -85,B 0,C 180,E1 -6885.543,E2 -6885.543} C_VEL
LIN {X 0,Y 481.66,Z 411.49,A -85,B 0,C 180,E1 -6888.958,E2 -6888.958} C_VEL
LIN {X 0,Y 481.705,Z 411.61,A -85,B 0,C 180,E1 -6890.14,E2 -6890.14} C_VEL
LIN {X 0,Y 483.765,Z 421.989,A -85,B 0,C 180,E1 -6893.037,E2 -6893.037} C_VEL
LIN {X 0,Y 484.086,Z 425.623,A -85,B 0,C 180,E1 -6893.986,E2 -6893.986} C_VEL
LIN {X 0,Y 483.35,Z 439.959,A -85,B 0,C 180,E1 -6897.494,E2 -6897.494} C_VEL
LIN {X 0,Y 482.986,Z 451.037,A -85,B 0,C 180,E1 -6900.107,E2 -6900.107} C_VEL
LIN {X 0,Y 482.65,Z 463.267,A -85,B 0,C 180,E1 -6902.91,E2 -6902.91} C_VEL
LIN {X 0,Y 482.289,Z 476.706,A -85,B 0,C 180,E1 -6905.919,E2 -6905.919} C_VEL
LIN {X 0,Y 481.965,Z 490.45,A -85,B 0,C 180,E1 -6908.947,E2 -6908.947} C_VEL
LIN {X 0,Y 481.671,Z 506.186,A -85,B 0,C 180,E1 -6912.376,E2 -6912.376} C_VEL
LIN {X 0,Y 481.439,Z 518.323,A -85,B 0,C 180,E1 -6915.009,E2 -6915.009} C_VEL
LIN {X 0,Y 482.81,Z 533.26,A -85,B 0,C 180,E1 -6915.403,E2 -6915.403} C_VEL
LIN {X 0,Y 483.699,Z 539.793,A -85,B 0,C 180,E1 -6915.646,E2 -6915.646} C_VEL
LIN {X 0,Y 483.276,Z 551.933,A -85,B 0,C 180,E1 -6916.17,E2 -6916.17} C_VEL
LIN {X 0,Y 482.796,Z 564.258,A -85,B 0,C 180,E1 -6916.885,E2 -6916.885} C_VEL
LIN {X 0,Y 482.35,Z 575.223,A -85,B 0,C 180,E1 -6917.695,E2 -6917.695} C_VEL
LIN {X 0,Y 481.956,Z 585.614,A -85,B 0,C 180,E1 -6918.646,E2 -6918.646} C_VEL
LIN {X 0,Y 481.643,Z 594.973,A -85,B 0,C 180,E1 -6919.703,E2 -6919.703} C_VEL
